LIN {X 0,Y 356.725,Z 687.983,A -85,B 0,C 180,E1 -20964.366,E2 -20964.366} C_VEL
LIN {X 0,Y 356.606,Z 693.356,A -85,B 0,C 180,E1 -20966.058,E2 -20966.058} C_VEL
LIN {X 0,Y 356.565,Z 697.608,A -85,B 0,C 180,E1 -20967.748,E2 -20967.748} C_VEL
LIN {X 0,Y 356.535,Z 699.927,A -85,B 0,C 180,E1 -20968.874,E2 -20968.874} C_VEL
LIN {X 0,Y 356.536,Z 701.836,A -85,B 0,C 180,E1 -20970,E2 -20970} C_VEL
LIN {X 0,Y 356.433,Z 704.456,A -85,B 0,C 180,E1 -20972.252,E2 -20972.252} C_VEL
LIN {X 0,Y 356.57,Z 705.616,A -85,B 0,C 180,E1 -20974.507,E2 -20974.507} C_VEL
LIN {X 0,Y 357.041,Z 705.356,A -85,B 0,C 180,E1 -20976.76,E2 -20976.76} C_VEL
LIN {X 0,Y 357.878,Z 703.692,A -85,B 0,C 180,E1 -20979.008,E2 -20979.008} C_VEL
LIN {X 0,Y 359.272,Z 700.612,A -85,B 0,C 180,E1 -20981.242,E2 -20981.242} C_VEL
LIN {X 0,Y 361.39,Z 696.021,A -85,B 0,C 180,E1 -20983.449,E2 -20983.449} C_VEL
LIN {X 0,Y 363.566,Z 690.094,A -85,B 0,C 180,E1 -20985.572,E2 -20985.572} C_VEL
LIN {X 0,Y 366.275,Z 682.97,A -85,B 0,C 180,E1 -20987.529,E2 -20987.529} C_VEL
LIN {X 0,Y 369.393,Z 674.484,A -85,B 0,C 180,E1 -20989.38,E2 -20989.38} C_VEL
LIN {X 0,Y 372.33,Z 665.799,A -85,B 0,C 180,E1 -20990.943,E2 -20990.943} C_VEL
LIN {X 0,Y 375.647,Z 655.443,A -85,B 0,C 180,E1 -20992.473,E2 -20992.473} C_VEL
LIN {X 0,Y 378.991,Z 644.123,A -85,B 0,C 180,E1 -20993.847,E2 -20993.847} C_VEL
LIN {X 0,Y 382.256,Z 631.813,A -85,B 0,C 180,E1 -20995.071,E2 -20995.071} C_VEL
LIN {X 0,Y 385.528,Z 618.219,A -85,B 0,C 180,E1 -20996.141,E2 -20996.141} C_VEL
LIN {X 0,Y 388.246,Z 605.333,A -85,B 0,C 180,E1 -20996.955,E2 -20996.955} C_VEL
LIN {X 0,Y 390.754,Z 591.419,A -85,B 0,C 180,E1 -20997.634,E2 -20997.634} C_VEL
LIN {X 0,Y 393.434,Z 571.086,A -85,B 0,C 180,E1 -20998.368,E2 -20998.368} C_VEL
LIN {X 0,Y 403.498,Z 492.971,A -85,B 0,C 180,E1 -21000.927,E2 -21000.927} C_VEL
LIN {X 0,Y 404.111,Z 486.973,A -85,B 0,C 180,E1 -21001.172,E2 -21001.172} C_VEL
LIN {X 0,Y 404.64,Z 471.101,A -85,B 0,C 180,E1 -21002.091,E2 -21002.091} C_VEL
LIN {X 0,Y 404.733,Z 459.98,A -85,B 0,C 180,E1 -21002.845,E2 -21002.845} C_VEL
LIN {X 0,Y 404.527,Z 444.365,A -85,B 0,C 180,E1 -21004.083,E2 -21004.083} C_VEL
LIN {X 0,Y 404.479,Z 437.616,A -85,B 0,C 180,E1 -21004.712,E2 -21004.712} C_VEL
LIN {X 0,Y 406.141,Z 430.503,A -85,B 0,C 180,E1 -21005.594,E2 -21005.594} C_VEL
LIN {X 0,Y 406.191,Z 429.05,A -85,B 0,C 180,E1 -21005.895,E2 -21005.895} C_VEL
LIN {X 0,Y 404.475,Z 426.255,A -85,B 0,C 180,E1 -21007.309,E2 -21007.309} C_VEL
LIN {X 0,Y 403.004,Z 424.19,A -85,B 0,C 180,E1 -21008.734,E2 -21008.734} C_VEL
LIN {X 0,Y 401.778,Z 422.799,A -85,B 0,C 180,E1 -21010.169,E2 -21010.169} C_VEL
LIN {X 0,Y 400.85,Z 422.022,A -85,B 0,C 180,E1 -21011.606,E2 -21011.606} C_VEL
LIN {X 0,Y 399.918,Z 421.946,A -85,B 0,C 180,E1 -21014.102,E2 -21014.102} C_VEL
LIN {X 0,Y 399.591,Z 423.06,A -85,B 0,C 180,E1 -21015.946,E2 -21015.946} C_VEL
LIN {X 0,Y 399.519,Z 425.806,A -85,B 0,C 180,E1 -21018.224,E2 -21018.224} C_VEL
LIN {X 0,Y 399.657,Z 428.065,A -85,B 0,C 180,E1 -21019.574,E2 -21019.574} C_VEL
LIN {X 0,Y 399.882,Z 432.504,A -85,B 0,C 180,E1 -21021.546,E2 -21021.546} C_VEL
LIN {X 0,Y 399.989,Z 438.039,A -85,B 0,C 180,E1 -21023.459,E2 -21023.459} C_VEL
LIN {X 0,Y 400.19,Z 440.153,A -85,B 0,C 180,E1 -21024.049,E2 -21024.049} C_VEL
LIN {X 0,Y 400.823,Z 442.858,A -85,B 0,C 180,E1 -21024.526,E2 -21024.526} C_VEL
LIN {X 0,Y 401.862,Z 457.626,A -85,B 0,C 180,E1 -21026.099,E2 -21026.099} C_VEL
LIN {X 0,Y 402.903,Z 473.385,A -85,B 0,C 180,E1 -21027.548,E2 -21027.548} C_VEL
LIN {X 0,Y 403.63,Z 486.988,A -85,B 0,C 180,E1 -21028.627,E2 -21028.627} C_VEL
LIN {X 0,Y 403.698,Z 493.511,A -85,B 0,C 180,E1 -21029.053,E2 -21029.053} C_VEL
LIN {X 0,Y 391.952,Z 585.206,A -85,B 0,C 180,E1 -21032.06,E2 -21032.06} C_VEL
LIN {X 0,Y 389.322,Z 600.595,A -85,B 0,C 180,E1 -21032.764,E2 -21032.764} C_VEL
LIN {X 0,Y 386.45,Z 614.844,A -85,B 0,C 180,E1 -21033.637,E2 -21033.637} C_VEL
LIN {X 0,Y 383.155,Z 628.608,A -85,B 0,C 180,E1 -21034.703,E2 -21034.703} C_VEL
LIN {X 0,Y 379.567,Z 642.265,A -85,B 0,C 180,E1 -21036.047,E2 -21036.047} C_VEL
LIN {X 0,Y 375.891,Z 654.552,A -85,B 0,C 180,E1 -21037.542,E2 -21037.542} C_VEL
LIN {X 0,Y 372.598,Z 664.764,A -85,B 0,C 180,E1 -21039.073,E2 -21039.073} C_VEL
LIN {X 0,Y 369.59,Z 673.378,A -85,B 0,C 180,E1 -21040.631,E2 -21040.631} C_VEL
LIN {X 0,Y 366.564,Z 681.749,A -85,B 0,C 180,E1 -21042.485,E2 -21042.485} C_VEL
LIN {X 0,Y 363.94,Z 688.565,A -85,B 0,C 180,E1 -21044.369,E2 -21044.369} C_VEL
LIN {X 0,Y 361.633,Z 694.693,A -85,B 0,C 180,E1 -21046.56,E2 -21046.56} C_VEL
LIN {X 0,Y 359.451,Z 699.244,A -85,B 0,C 180,E1 -21048.763,E2 -21048.763} C_VEL
LIN {X 0,Y 358.038,Z 702.291,A -85,B 0,C 180,E1 -21050.996,E2 -21050.996} C_VEL
LIN {X 0,Y 357.088,Z 703.936,A -85,B 0,C 180,E1 -21053.241,E2 -21053.241} C_VEL
LIN {X 0,Y 356.569,Z 704.185,A -85,B 0,C 180,E1 -21055.494,E2 -21055.494} C_VEL
LIN {X 0,Y 356.377,Z 703.027,A -85,B 0,C 180,E1 -21057.747,E2 -21057.747} C_VEL
LIN {X 0,Y 356.436,Z 700.429,A -85,B 0,C 180,E1 -21060,E2 -21060} C_VEL
LIN {X 0,Y 356.48,Z 696.249,A -85,B 0,C 180,E1 -21062.252,E2 -21062.252} C_VEL
LIN {X 0,Y 356.556,Z 692.048,A -85,B 0,C 180,E1 -21063.943,E2 -21063.943} C_VEL
LIN {X 0,Y 356.686,Z 685.768,A -85,B 0,C 180,E1 -21065.918,E2 -21065.918} C_VEL
LIN {X 0,Y 356.95,Z 677.854,A -85,B 0,C 180,E1 -21067.896,E2 -21067.896} C_VEL
LIN {X 0,Y 357.418,Z 669.599,A -85,B 0,C 180,E1 -21069.589,E2 -21069.589} C_VEL
LIN {X 0,Y 357.937,Z 659.637,A -85,B 0,C 180,E1 -21071.285,E2 -21071.285} C_VEL
LIN {X 0,Y 358.682,Z 648.682,A -85,B 0,C 180,E1 -21072.835,E2 -21072.835} C_VEL
LIN {X 0,Y 359.384,Z 636.555,A -85,B 0,C 180,E1 -21074.245,E2 -21074.245} C_VEL
LIN {X 0,Y 360.308,Z 623.272,A -85,B 0,C 180,E1 -21075.504,E2 -21075.504} C_VEL
LIN {X 0,Y 361.095,Z 609.51,A -85,B 0,C 180,E1 -21076.554,E2 -21076.554} C_VEL
LIN {X 0,Y 361.848,Z 594.748,A -85,B 0,C 180,E1 -21077.424,E2 -21077.424} C_VEL
LIN {X 0,Y 362.486,Z 579.344,A -85,B 0,C 180,E1 -21078.083,E2 -21078.083} C_VEL
LIN {X 0,Y 365.761,Z 475.035,A -85,B 0,C 180,E1 -21081.209,E2 -21081.209} C_VEL
LIN {X 0,Y 363.266,Z 445.339,A -85,B 0,C 180,E1 -21082.179,E2 -21082.179} C_VEL
LIN {X 0,Y 363.025,Z 439.566,A -85,B 0,C 180,E1 -21082.376,E2 -21082.376} C_VEL
LIN {X 0,Y 365.15,Z 412.697,A -85,B 0,C 180,E1 -21086.181,E2 -21086.181} C_VEL
LIN {X 0,Y 367.059,Z 389.753,A -85,B 0,C 180,E1 -21089.432,E2 -21089.432} C_VEL
LIN {X 0,Y 363.105,Z 371.527,A -85,B 0,C 180,E1 -21092.275,E2 -21092.275} C_VEL
LIN {X 0,Y 359.011,Z 353.326,A -85,B 0,C 180,E1 -21095.234,E2 -21095.234} C_VEL
LIN {X 0,Y 358.937,Z 353.332,A -85,B 0,C 180,E1 -21098.687,E2 -21098.687} C_VEL
LIN {X 0,Y 358.948,Z 353.327,A -85,B 0,C 180,E1 -21102.139,E2 -21102.139} C_VEL
LIN {X 0,Y 358.972,Z 353.324,A -85,B 0,C 180,E1 -21105.376,E2 -21105.376} C_VEL
LIN {X 0,Y 358.95,Z 353.33,A -85,B 0,C 180,E1 -21108.435,E2 -21108.435} C_VEL
LIN {X 0,Y 358.943,Z 353.33,A -85,B 0,C 180,E1 -21111.358,E2 -21111.358} C_VEL
LIN {X 0,Y 358.964,Z 353.328,A -85,B 0,C 180,E1 -21115.04,E2 -21115.04} C_VEL
LIN {X 0,Y 358.978,Z 353.321,A -85,B 0,C 180,E1 -21119.154,E2 -21119.154} C_VEL
LIN {X 0,Y 358.971,Z 353.327,A -85,B 0,C 180,E1 -21122.076,E2 -21122.076} C_VEL
LIN {X 0,Y 358.971,Z 353.329,A -85,B 0,C 180,E1 -21124.578,E2 -21124.578} C_VEL
LIN {X 0,Y 358.986,Z 353.325,A -85,B 0,C 180,E1 -21127.031,E2 -21127.031} C_VEL
LIN {X 0,Y 359.04,Z 353.321,A -85,B 0,C 180,E1 -21129.68,E2 -21129.68} C_VEL
LIN {X 0,Y 360.677,Z 357.57,A -85,B 0,C 180,E1 -21129.891,E2 -21129.891} C_VEL
LIN {X 0,Y 369.779,Z 378.619,A -85,B 0,C 180,E1 -21130.947,E2 -21130.947} C_VEL
LIN {X 0,Y 372.167,Z 384.575,A -85,B 0,C 180,E1 -21131.223,E2 -21131.223} C_VEL
LIN {X 0,Y 371.034,Z 437.953,A -85,B 0,C 180,E1 -21132.243,E2 -21132.243} C_VEL
LIN {X 0,Y 370.729,Z 471.673,A -85,B 0,C 180,E1 -21132.936,E2 -21132.936} C_VEL
LIN {X 0,Y 370.297,Z 486.255,A -85,B 0,C 180,E1 -21133.446,E2 -21133.446} C_VEL
LIN {X 0,Y 369.662,Z 499.54,A -85,B 0,C 180,E1 -21134.124,E2 -21134.124} C_VEL
LIN {X 0,Y 368.668,Z 512.538,A -85,B 0,C 180,E1 -21134.997,E2 -21134.997} C_VEL
LIN {X 0,Y 367.573,Z 525.068,A -85,B 0,C 180,E1 -21136.079,E2 -21136.079} C_VEL
LIN {X 0,Y 366.34,Z 537.468,A -85,B 0,C 180,E1 -21137.42,E2 -21137.42} C_VEL
LIN {X 0,Y 365.038,Z 546.962,A -85,B 0,C 180,E1 -21138.657,E2 -21138.657} C_VEL
LIN {X 0,Y 363.495,Z 557.369,A -85,B 0,C 180,E1 -21140.293,E2 -21140.293} C_VEL
LIN {X 0,Y 362.248,Z 565.948,A -85,B 0,C 180,E1 -21141.942,E2 -21141.942} C_VEL
LIN {X 0,Y 361.022,Z 574.183,A -85,B 0,C 180,E1 -21143.874,E2 -21143.874} C_VEL
LIN {X 0,Y 360.094,Z 579.941,A -85,B 0,C 180,E1 -21145.538,E2 -21145.538} C_VEL
LIN {X 0,Y 359.226,Z 586.093,A -85,B 0,C 180,E1 -21147.765,E2 -21147.765} C_VEL
LIN {X 0,Y 358.678,Z 590.642,A -85,B 0,C 180,E1 -21150,E2 -21150} C_VEL
LIN {X 0,Y 358.344,Z 593.75,A -85,B 0,C 180,E1 -21152.241,E2 -21152.241} C_VEL
LIN {X 0,Y 358.327,Z 595.525,A -85,B 0,C 180,E1 -21154.485,E2 -21154.485} C_VEL
LIN {X 0,Y 358.461,Z 596.018,A -85,B 0,C 180,E1 -21156.733,E2 -21156.733} C_VEL
LIN {X 0,Y 358.889,Z 595.216,A -85,B 0,C 180,E1 -21158.983,E2 -21158.983} C_VEL
LIN {X 0,Y 359.497,Z 593.109,A -85,B 0,C 180,E1 -21161.236,E2 -21161.236} C_VEL
LIN {X 0,Y 360.637,Z 589.599,A -85,B 0,C 180,E1 -21163.478,E2 -21163.478} C_VEL
LIN {X 0,Y 361.996,Z 584.607,A -85,B 0,C 180,E1 -21165.718,E2 -21165.718} C_VEL
LIN {X 0,Y 363.238,Z 579.74,A -85,B 0,C 180,E1 -21167.391,E2 -21167.391} C_VEL
LIN {X 0,Y 364.927,Z 572.832,A -85,B 0,C 180,E1 -21169.311,E2 -21169.311} C_VEL
LIN {X 0,Y 366.614,Z 565.377,A -85,B 0,C 180,E1 -21170.992,E2 -21170.992} C_VEL
LIN {X 0,Y 368.514,Z 556.498,A -85,B 0,C 180,E1 -21172.638,E2 -21172.638} C_VEL
LIN {X 0,Y 370.572,Z 545.708,A -85,B 0,C 180,E1 -21174.275,E2 -21174.275} C_VEL
LIN {X 0,Y 372.362,Z 534.709,A -85,B 0,C 180,E1 -21175.636,E2 -21175.636} C_VEL
LIN {X 0,Y 374.154,Z 522.52,A -85,B 0,C 180,E1 -21176.849,E2 -21176.849} C_VEL
LIN {X 0,Y 375.546,Z 510.75,A -85,B 0,C 180,E1 -21177.794,E2 -21177.794} C_VEL
LIN {X 0,Y 376.487,Z 499.1,A -85,B 0,C 180,E1 -21178.549,E2 -21178.549} C_VEL
LIN {X 0,Y 377.342,Z 484.813,A -85,B 0,C 180,E1 -21179.241,E2 -21179.241} C_VEL
LIN {X 0,Y 377.785,Z 470.873,A -85,B 0,C 180,E1 -21179.698,E2 -21179.698} C_VEL
LIN {X 0,Y 379.518,Z 405.514,A -85,B 0,C 180,E1 -21180.954,E2 -21180.954} C_VEL
LIN {X 0,Y 379.586,Z 394.59,A -85,B 0,C 180,E1 -21181.18,E2 -21181.18} C_VEL
LIN {X 0,Y 370.189,Z 374.863,A -85,B 0,C 180,E1 -21182.424,E2 -21182.424} C_VEL
LIN {X 0,Y 360.343,Z 356.812,A -85,B 0,C 180,E1 -21183.757,E2 -21183.757} C_VEL
LIN {X 0,Y 359.066,Z 354.304,A -85,B 0,C 180,E1 -21183.941,E2 -21183.941} C_VEL
LIN {X 0,Y 358.893,Z 353.337,A -85,B 0,C 180,E1 -21184.001,E2 -21184.001} C_VEL
LIN {X 0,Y 358.912,Z 353.335,A -85,B 0,C 180,E1 -21187.228,E2 -21187.228} C_VEL
LIN {X 0,Y 358.912,Z 353.338,A -85,B 0,C 180,E1 -21190.437,E2 -21190.437} C_VEL
LIN {X 0,Y 358.886,Z 353.338,A -85,B 0,C 180,E1 -21191.966,E2 -21191.966} C_VEL
LIN {X 0,Y 358.237,Z 353.422,A -85,B 0,C 180,E1 -21192.901,E2 -21192.901} C_VEL
LIN {X 0,Y 355.372,Z 353.774,A -85,B 0,C 180,E1 -21194.422,E2 -21194.422} C_VEL
LIN {X 0,Y 352.944,Z 354.077,A -85,B 0,C 180,E1 -21195.653,E2 -21195.653} C_VEL
LIN {X 0,Y 351.92,Z 354.207,A -85,B 0,C 180,E1 -21196.606,E2 -21196.606} C_VEL
LIN {X 0,Y 351.848,Z 354.209,A -85,B 0,C 180,E1 -21196.929,E2 -21196.929} C_VEL
LIN {X 0,Y 351.854,Z 354.209,A -85,B 0,C 180,E1 -21200.429,E2 -21200.429} C_VEL
LIN {X 0,Y 351.864,Z 354.168,A -85,B 0,C 180,E1 -21203.33,E2 -21203.33} C_VEL
LIN {X 0,Y 351.865,Z 354.208,A -85,B 0,C 180,E1 -21206.729,E2 -21206.729} C_VEL
LIN {X 0,Y 351.886,Z 354.2,A -85,B 0,C 180,E1 -21210.156,E2 -21210.156} C_VEL
LIN {X 0,Y 351.946,Z 354.189,A -85,B 0,C 180,E1 -21214.033,E2 -21214.033} C_VEL
LIN {X 0,Y 351.954,Z 354.198,A -85,B 0,C 180,E1 -21217.572,E2 -21217.572} C_VEL
LIN {X 0,Y 358.141,Z 377.526,A -85,B 0,C 180,E1 -21218.454,E2 -21218.454} C_VEL
LIN {X 0,Y 355.675,Z 470.004,A -85,B 0,C 180,E1 -21221.237,E2 -21221.237} C_VEL
LIN {X 0,Y 355.334,Z 485.438,A -85,B 0,C 180,E1 -21221.912,E2 -21221.912} C_VEL
LIN {X 0,Y 354.727,Z 501.095,A -85,B 0,C 180,E1 -21222.845,E2 -21222.845} C_VEL
LIN {X 0,Y 354.11,Z 514.993,A -85,B 0,C 180,E1 -21223.923,E2 -21223.923} C_VEL
LIN {X 0,Y 353.351,Z 528.412,A -85,B 0,C 180,E1 -21225.213,E2 -21225.213} C_VEL
LIN {X 0,Y 352.707,Z 540.9,A -85,B 0,C 180,E1 -21226.681,E2 -21226.681} C_VEL
LIN {X 0,Y 352.08,Z 551.828,A -85,B 0,C 180,E1 -21228.233,E2 -21228.233} C_VEL
LIN {X 0,Y 351.512,Z 561.982,A -85,B 0,C 180,E1 -21229.958,E2 -21229.958} C_VEL
LIN {X 0,Y 351.108,Z 570.476,A -85,B 0,C 180,E1 -21231.684,E2 -21231.684} C_VEL
LIN {X 0,Y 350.843,Z 578.663,A -85,B 0,C 180,E1 -21233.696,E2 -21233.696} C_VEL
LIN {X 0,Y 350.805,Z 584.378,A -85,B 0,C 180,E1 -21235.419,E2 -21235.419} C_VEL
LIN {X 0,Y 350.847,Z 589.454,A -85,B 0,C 180,E1 -21237.294,E2 -21237.294} C_VEL
LIN {X 0,Y 351.077,Z 593.911,A -85,B 0,C 180,E1 -21239.428,E2 -21239.428} C_VEL
LIN {X 0,Y 351.487,Z 596.487,A -85,B 0,C 180,E1 -21241.142,E2 -21241.142} C_VEL
LIN {X 0,Y 352.352,Z 598.709,A -85,B 0,C 180,E1 -21243.419,E2 -21243.419} C_VEL
LIN {X 0,Y 353.573,Z 599.494,A -85,B 0,C 180,E1 -21245.684,E2 -21245.684} C_VEL
LIN {X 0,Y 355.059,Z 598.85,A -85,B 0,C 180,E1 -21247.937,E2 -21247.937} C_VEL
LIN {X 0,Y 357.111,Z 596.776,A -85,B 0,C 180,E1 -21250.167,E2 -21250.167} C_VEL
LIN {X 0,Y 359.825,Z 593.175,A -85,B 0,C 180,E1 -21252.364,E2 -21252.364} C_VEL
LIN {X 0,Y 361.983,Z 589.458,A -85,B 0,C 180,E1 -21253.997,E2 -21253.997} C_VEL
LIN {X 0,Y 365.123,Z 583.078,A -85,B 0,C 180,E1 -21256.15,E2 -21256.15} C_VEL
LIN {X 0,Y 368.201,Z 575.99,A -85,B 0,C 180,E1 -21257.978,E2 -21257.978} C_VEL
LIN {X 0,Y 371.607,Z 566.998,A -85,B 0,C 180,E1 -21259.833,E2 -21259.833} C_VEL
LIN {X 0,Y 374.756,Z 557.748,A -85,B 0,C 180,E1 -21261.375,E2 -21261.375} C_VEL
LIN {X 0,Y 378.134,Z 546.581,A -85,B 0,C 180,E1 -21262.892,E2 -21262.892} C_VEL
LIN {X 0,Y 381.462,Z 534.045,A -85,B 0,C 180,E1 -21264.258,E2 -21264.258} C_VEL
LIN {X 0,Y 384.193,Z 521.641,A -85,B 0,C 180,E1 -21265.368,E2 -21265.368} C_VEL
LIN {X 0,Y 386.585,Z 508.111,A -85,B 0,C 180,E1 -21266.353,E2 -21266.353} C_VEL
LIN {X 0,Y 388.641,Z 493.528,A -85,B 0,C 180,E1 -21267.179,E2 -21267.179} C_VEL
LIN {X 0,Y 390.48,Z 476.072,A -85,B 0,C 180,E1 -21267.909,E2 -21267.909} C_VEL
LIN {X 0,Y 394.84,Z 439.615,A -85,B 0,C 180,E1 -21269.138,E2 -21269.138} C_VEL
LIN {X 0,Y 397.763,Z 417.256,A -85,B 0,C 180,E1 -21269.877,E2 -21269.877} C_VEL
LIN {X 0,Y 394.545,Z 410.848,A -85,B 0,C 180,E1 -21271.112,E2 -21271.112} C_VEL
LIN {X 0,Y 391.131,Z 404.658,A -85,B 0,C 180,E1 -21272.567,E2 -21272.567} C_VEL
LIN {X 0,Y 389.244,Z 401.397,A -85,B 0,C 180,E1 -21273.486,E2 -21273.486} C_VEL
LIN {X 0,Y 386.985,Z 397.73,A -85,B 0,C 180,E1 -21274.686,E2 -21274.686} C_VEL
LIN {X 0,Y 384.579,Z 393.864,A -85,B 0,C 180,E1 -21276.183,E2 -21276.183} C_VEL
LIN {X 0,Y 382.361,Z 390.848,A -85,B 0,C 180,E1 -21277.858,E2 -21277.858} C_VEL
LIN {X 0,Y 381.655,Z 389.329,A -85,B 0,C 180,E1 -21278.608,E2 -21278.608} C_VEL
LIN {X 0,Y 379.403,Z 387.476,A -85,B 0,C 180,E1 -21281.653,E2 -21281.653} C_VEL
LIN {X 0,Y 379.063,Z 387.134,A -85,B 0,C 180,E1 -21283.891,E2 -21283.891} C_VEL
LIN {X 0,Y 379.695,Z 387.952,A -85,B 0,C 180,E1 -21286.009,E2 -21286.009} C_VEL
LIN {X 0,Y 381.505,Z 389.601,A -85,B 0,C 180,E1 -21288.266,E2 -21288.266} C_VEL
LIN {X 0,Y 383.095,Z 392.706,A -85,B 0,C 180,E1 -21289.849,E2 -21289.849} C_VEL
LIN {X 0,Y 384.649,Z 394.585,A -85,B 0,C 180,E1 -21290.94,E2 -21290.94} C_VEL
LIN {X 0,Y 385.11,Z 396.18,A -85,B 0,C 180,E1 -21291.344,E2 -21291.344} C_VEL
LIN {X 0,Y 386.64,Z 403.777,A -85,B 0,C 180,E1 -21292.794,E2 -21292.794} C_VEL
LIN {X 0,Y 389.443,Z 417.992,A -85,B 0,C 180,E1 -21294.984,E2 -21294.984} C_VEL
LIN {X 0,Y 389.605,Z 422.458,A -85,B 0,C 180,E1 -21295.388,E2 -21295.388} C_VEL
LIN {X 0,Y 390.1,Z 441.215,A -85,B 0,C 180,E1 -21296.884,E2 -21296.884} C_VEL
LIN {X 0,Y 390.469,Z 462.05,A -85,B 0,C 180,E1 -21298.323,E2 -21298.323} C_VEL
LIN {X 0,Y 390.358,Z 475.663,A -85,B 0,C 180,E1 -21299.13,E2 -21299.13} C_VEL
LIN {X 0,Y 389.701,Z 489.992,A -85,B 0,C 180,E1 -21299.817,E2 -21299.817} C_VEL
LIN {X 0,Y 383.661,Z 539.895,A -85,B 0,C 180,E1 -21301.475,E2 -21301.475} C_VEL
LIN {X 0,Y 380.891,Z 555.484,A -85,B 0,C 180,E1 -21302.146,E2 -21302.146} C_VEL
LIN {X 0,Y 377.711,Z 570.021,A -85,B 0,C 180,E1 -21302.977,E2 -21302.977} C_VEL
LIN {X 0,Y 373.554,Z 586.152,A -85,B 0,C 180,E1 -21304.153,E2 -21304.153} C_VEL
LIN {X 0,Y 369.789,Z 599.191,A -85,B 0,C 180,E1 -21305.372,E2 -21305.372} C_VEL
LIN {X 0,Y 366.374,Z 610.138,A -85,B 0,C 180,E1 -21306.627,E2 -21306.627} C_VEL
LIN {X 0,Y 362.633,Z 621.676,A -85,B 0,C 180,E1 -21308.234,E2 -21308.234} C_VEL
LIN {X 0,Y 359.212,Z 632.199,A -85,B 0,C 180,E1 -21310.047,E2 -21310.047} C_VEL
LIN {X 0,Y 356.141,Z 641.2,A -85,B 0,C 180,E1 -21311.955,E2 -21311.955} C_VEL
LIN {X 0,Y 353.827,Z 648.647,A -85,B 0,C 180,E1 -21313.91,E2 -21313.91} C_VEL
LIN {X 0,Y 351.965,Z 655.474,A -85,B 0,C 180,E1 -21316.183,E2 -21316.183} C_VEL
LIN {X 0,Y 350.749,Z 660.764,A -85,B 0,C 180,E1 -21318.48,E2 -21318.48} C_VEL
LIN {X 0,Y 350.609,Z 661.973,A -85,B 0,C 180,E1 -21319.059,E2 -21319.059} C_VEL
LIN {X 0,Y 350.177,Z 671.911,A -85,B 0,C 180,E1 -21320.792,E2 -21320.792} C_VEL
LIN {X 0,Y 349.799,Z 680.094,A -85,B 0,C 180,E1 -21322.521,E2 -21322.521} C_VEL
LIN {X 0,Y 349.661,Z 686.861,A -85,B 0,C 180,E1 -21324.251,E2 -21324.251} C_VEL
LIN {X 0,Y 349.56,Z 692.399,A -85,B 0,C 180,E1 -21325.978,E2 -21325.978} C_VEL
LIN {X 0,Y 349.498,Z 696.863,A -85,B 0,C 180,E1 -21327.703,E2 -21327.703} C_VEL
LIN {X 0,Y 349.454,Z 700.358,A -85,B 0,C 180,E1 -21329.426,E2 -21329.426} C_VEL
LIN {X 0,Y 349.373,Z 702.903,A -85,B 0,C 180,E1 -21331.149,E2 -21331.149} C_VEL
LIN {X 0,Y 349.378,Z 705.024,A -85,B 0,C 180,E1 -21333.448,E2 -21333.448} C_VEL
LIN {X 0,Y 349.708,Z 705.692,A -85,B 0,C 180,E1 -21335.747,E2 -21335.747} C_VEL
LIN {X 0,Y 350.41,Z 704.936,A -85,B 0,C 180,E1 -21338.043,E2 -21338.043} C_VEL
LIN {X 0,Y 351.518,Z 702.787,A -85,B 0,C 180,E1 -21340.331,E2 -21340.331} C_VEL
LIN {X 0,Y 353.358,Z 699.197,A -85,B 0,C 180,E1 -21342.594,E2 -21342.594} C_VEL
LIN {X 0,Y 355.677,Z 694.096,A -85,B 0,C 180,E1 -21344.833,E2 -21344.833} C_VEL
LIN {X 0,Y 357.621,Z 689.234,A -85,B 0,C 180,E1 -21346.499,E2 -21346.499} C_VEL
LIN {X 0,Y 360.976,Z 681.121,A -85,B 0,C 180,E1 -21348.673,E2 -21348.673} C_VEL
LIN {X 0,Y 364.363,Z 672.316,A -85,B 0,C 180,E1 -21350.538,E2 -21350.538} C_VEL
LIN {X 0,Y 367.641,Z 663.241,A -85,B 0,C 180,E1 -21352.104,E2 -21352.104} C_VEL
LIN {X 0,Y 371.549,Z 651.413,A -85,B 0,C 180,E1 -21353.763,E2 -21353.763} C_VEL
LIN {X 0,Y 375.196,Z 639.346,A -85,B 0,C 180,E1 -21355.133,E2 -21355.133} C_VEL
LIN {X 0,Y 378.422,Z 627.589,A -85,B 0,C 180,E1 -21356.226,E2 -21356.226} C_VEL
LIN {X 0,Y 381.863,Z 613.173,A -85,B 0,C 180,E1 -21357.295,E2 -21357.295} C_VEL
LIN {X 0,Y 385.061,Z 597.984,A -85,B 0,C 180,E1 -21358.152,E2 -21358.152} C_VEL
LIN {X 0,Y 387.515,Z 583.341,A -85,B 0,C 180,E1 -21358.767,E2 -21358.767} C_VEL
LIN {X 0,Y 399.954,Z 491.497,A -85,B 0,C 180,E1 -21361.846,E2 -21361.846} C_VEL
LIN {X 0,Y 400.582,Z 481.749,A -85,B 0,C 180,E1 -21362.367,E2 -21362.367} C_VEL
LIN {X 0,Y 401.101,Z 466.574,A -85,B 0,C 180,E1 -21363.339,E2 -21363.339} C_VEL
LIN {X 0,Y 401.201,Z 449.322,A -85,B 0,C 180,E1 -21364.695,E2 -21364.695} C_VEL
LIN {X 0,Y 401.22,Z 437.905,A -85,B 0,C 180,E1 -21365.776,E2 -21365.776} C_VEL
LIN {X 0,Y 401.735,Z 435.888,A -85,B 0,C 180,E1 -21366.039,E2 -21366.039} C_VEL
LIN {X 0,Y 401.941,Z 434.259,A -85,B 0,C 180,E1 -21366.335,E2 -21366.335} C_VEL
LIN {X 0,Y 400.008,Z 431.305,A -85,B 0,C 180,E1 -21368.003,E2 -21368.003} C_VEL
LIN {X 0,Y 398.697,Z 429.59,A -85,B 0,C 180,E1 -21369.375,E2 -21369.375} C_VEL
LIN {X 0,Y 397.615,Z 428.454,A -85,B 0,C 180,E1 -21370.756,E2 -21370.756} C_VEL
LIN {X 0,Y 396.75,Z 427.877,A -85,B 0,C 180,E1 -21372.142,E2 -21372.142} C_VEL
LIN {X 0,Y 396.126,Z 427.794,A -85,B 0,C 180,E1 -21373.599,E2 -21373.599} C_VEL
LIN {X 0,Y 395.735,Z 428.344,A -85,B 0,C 180,E1 -21375.072,E2 -21375.072} C_VEL
LIN {X 0,Y 395.476,Z 429.583,A -85,B 0,C 180,E1 -21376.566,E2 -21376.566} C_VEL
LIN {X 0,Y 395.364,Z 432.992,A -85,B 0,C 180,E1 -21379.042,E2 -21379.042} C_VEL
LIN {X 0,Y 395.429,Z 437.508,A -85,B 0,C 180,E1 -21381.205,E2 -21381.205} C_VEL
LIN {X 0,Y 395.627,Z 440.106,A -85,B 0,C 180,E1 -21382.136,E2 -21382.136} C_VEL
LIN {X 0,Y 397.718,Z 446.772,A -85,B 0,C 180,E1 -21383.775,E2 -21383.775} C_VEL
LIN {X 0,Y 398.279,Z 457.122,A -85,B 0,C 180,E1 -21384.94,E2 -21384.94} C_VEL
LIN {X 0,Y 399.104,Z 473.805,A -85,B 0,C 180,E1 -21386.57,E2 -21386.57} C_VEL
LIN {X 0,Y 399.675,Z 488.703,A -85,B 0,C 180,E1 -21387.798,E2 -21387.798} C_VEL
LIN {X 0,Y 399.696,Z 495.123,A -85,B 0,C 180,E1 -21388.24,E2 -21388.24} C_VEL
LIN {X 0,Y 387.55,Z 584.975,A -85,B 0,C 180,E1 -21391.236,E2 -21391.236} C_VEL
LIN {X 0,Y 384.897,Z 599.742,A -85,B 0,C 180,E1 -21391.909,E2 -21391.909} C_VEL
LIN {X 0,Y 382.031,Z 613.198,A -85,B 0,C 180,E1 -21392.718,E2 -21392.718} C_VEL
LIN {X 0,Y 378.607,Z 627.223,A -85,B 0,C 180,E1 -21393.788,E2 -21393.788} C_VEL
LIN {X 0,Y 375.071,Z 639.894,A -85,B 0,C 180,E1 -21395.006,E2 -21395.006} C_VEL
LIN {X 0,Y 371.498,Z 651.579,A -85,B 0,C 180,E1 -21396.381,E2 -21396.381} C_VEL
LIN {X 0,Y 367.889,Z 662.278,A -85,B 0,C 180,E1 -21397.912,E2 -21397.912} C_VEL
LIN {X 0,Y 364.636,Z 671.25,A -85,B 0,C 180,E1 -21399.478,E2 -21399.478} C_VEL
LIN {X 0,Y 361.278,Z 679.963,A -85,B 0,C 180,E1 -21401.343,E2 -21401.343} C_VEL
LIN {X 0,Y 358.718,Z 686.184,A -85,B 0,C 180,E1 -21402.969,E2 -21402.969} C_VEL
LIN {X 0,Y 356.487,Z 691.34,A -85,B 0,C 180,E1 -21404.618,E2 -21404.618} C_VEL
LIN {X 0,Y 354.167,Z 696.786,A -85,B 0,C 180,E1 -21406.854,E2 -21406.854} C_VEL
LIN {X 0,Y 352.531,Z 699.841,A -85,B 0,C 180,E1 -21408.54,E2 -21408.54} C_VEL
LIN {X 0,Y 351.022,Z 702.673,A -85,B 0,C 180,E1 -21410.815,E2 -21410.815} C_VEL
LIN {X 0,Y 350.039,Z 704.106,A -85,B 0,C 180,E1 -21413.105,E2 -21413.105} C_VEL
LIN {X 0,Y 349.483,Z 704.148,A -85,B 0,C 180,E1 -21415.402,E2 -21415.402} C_VEL
LIN {X 0,Y 349.291,Z 702.764,A -85,B 0,C 180,E1 -21417.702,E2 -21417.702} C_VEL
LIN {X 0,Y 349.356,Z 699.926,A -85,B 0,C 180,E1 -21420,E2 -21420} C_VEL
LIN {X 0,Y 349.395,Z 696.826,A -85,B 0,C 180,E1 -21421.724,E2 -21421.724} C_VEL
LIN {X 0,Y 349.442,Z 692.719,A -85,B 0,C 180,E1 -21423.448,E2 -21423.448} C_VEL
LIN {X 0,Y 349.57,Z 687.607,A -85,B 0,C 180,E1 -21425.174,E2 -21425.174} C_VEL
LIN {X 0,Y 349.81,Z 680.21,A -85,B 0,C 180,E1 -21427.19,E2 -21427.19} C_VEL
LIN {X 0,Y 350.123,Z 672.424,A -85,B 0,C 180,E1 -21428.92,E2 -21428.92} C_VEL
LIN {X 0,Y 350.669,Z 663.069,A -85,B 0,C 180,E1 -21430.648,E2 -21430.648} C_VEL
LIN {X 0,Y 351.368,Z 652.325,A -85,B 0,C 180,E1 -21432.29,E2 -21432.29} C_VEL
LIN {X 0,Y 352.098,Z 640.244,A -85,B 0,C 180,E1 -21433.811,E2 -21433.811} C_VEL
LIN {X 0,Y 352.88,Z 627.823,A -85,B 0,C 180,E1 -21435.101,E2 -21435.101} C_VEL
LIN {X 0,Y 353.786,Z 614.357,A -85,B 0,C 180,E1 -21436.24,E2 -21436.24} C_VEL
LIN {X 0,Y 354.433,Z 600.335,A -85,B 0,C 180,E1 -21437.17,E2 -21437.17} C_VEL
LIN {X 0,Y 355.117,Z 585.482,A -85,B 0,C 180,E1 -21437.914,E2 -21437.914} C_VEL
LIN {X 0,Y 355.72,Z 568.346,A -85,B 0,C 180,E1 -21438.508,E2 -21438.508} C_VEL
LIN {X 0,Y 358.743,Z 475.397,A -85,B 0,C 180,E1 -21441.363,E2 -21441.363} C_VEL
LIN {X 0,Y 356.26,Z 445.66,A -85,B 0,C 180,E1 -21442.355,E2 -21442.355} C_VEL
LIN {X 0,Y 356.016,Z 439.606,A -85,B 0,C 180,E1 -21442.563,E2 -21442.563} C_VEL
LIN {X 0,Y 358.22,Z 412.54,A -85,B 0,C 180,E1 -21446.448,E2 -21446.448} C_VEL
LIN {X 0,Y 360.065,Z 390.739,A -85,B 0,C 180,E1 -21449.58,E2 -21449.58} C_VEL
LIN {X 0,Y 355.778,Z 371.172,A -85,B 0,C 180,E1 -21452.684,E2 -21452.684} C_VEL
LIN {X 0,Y 351.972,Z 354.202,A -85,B 0,C 180,E1 -21455.453,E2 -21455.453} C_VEL
LIN {X 0,Y 351.874,Z 354.214,A -85,B 0,C 180,E1 -21459.074,E2 -21459.074} C_VEL
LIN {X 0,Y 351.923,Z 354.203,A -85,B 0,C 180,E1 -21462.588,E2 -21462.588} C_VEL
LIN {X 0,Y 351.939,Z 354.198,A -85,B 0,C 180,E1 -21465.846,E2 -21465.846} C_VEL
LIN {X 0,Y 351.882,Z 354.206,A -85,B 0,C 180,E1 -21469.15,E2 -21469.15} C_VEL
LIN {X 0,Y 351.914,Z 354.205,A -85,B 0,C 180,E1 -21472.765,E2 -21472.765} C_VEL
LIN {X 0,Y 351.895,Z 354.207,A -85,B 0,C 180,E1 -21476.128,E2 -21476.128} C_VEL
LIN {X 0,Y 351.928,Z 354.201,A -85,B 0,C 180,E1 -21480.16,E2 -21480.16} C_VEL
LIN {X 0,Y 351.931,Z 354.203,A -85,B 0,C 180,E1 -21483.591,E2 -21483.591} C_VEL
LIN {X 0,Y 351.98,Z 354.201,A -85,B 0,C 180,E1 -21486.547,E2 -21486.547} C_VEL
LIN {X 0,Y 351.979,Z 354.2,A -85,B 0,C 180,E1 -21489.191,E2 -21489.191} C_VEL
LIN {X 0,Y 352.975,Z 357.048,A -85,B 0,C 180,E1 -21489.329,E2 -21489.329} C_VEL
LIN {X 0,Y 361.343,Z 375.884,A -85,B 0,C 180,E1 -21490.327,E2 -21490.327} C_VEL
LIN {X 0,Y 365.602,Z 386.378,A -85,B 0,C 180,E1 -21490.834,E2 -21490.834} C_VEL
LIN {X 0,Y 364.181,Z 459.074,A -85,B 0,C 180,E1 -21492.258,E2 -21492.258} C_VEL
LIN {X 0,Y 363.992,Z 476.544,A -85,B 0,C 180,E1 -21492.682,E2 -21492.682} C_VEL
LIN {X 0,Y 363.496,Z 490.484,A -85,B 0,C 180,E1 -21493.235,E2 -21493.235} C_VEL
LIN {X 0,Y 362.641,Z 504.553,A -85,B 0,C 180,E1 -21494.024,E2 -21494.024} C_VEL
LIN {X 0,Y 361.565,Z 517.456,A -85,B 0,C 180,E1 -21494.983,E2 -21494.983} C_VEL
LIN {X 0,Y 360.382,Z 530.434,A -85,B 0,C 180,E1 -21496.226,E2 -21496.226} C_VEL
LIN {X 0,Y 359.032,Z 542.099,A -85,B 0,C 180,E1 -21497.608,E2 -21497.608} C_VEL
LIN {X 0,Y 357.617,Z 551.792,A -85,B 0,C 180,E1 -21498.991,E2 -21498.991} C_VEL
LIN {X 0,Y 356.174,Z 561.456,A -85,B 0,C 180,E1 -21500.663,E2 -21500.663} C_VEL
LIN {X 0,Y 354.949,Z 569.479,A -85,B 0,C 180,E1 -21502.345,E2 -21502.345} C_VEL
LIN {X 0,Y 353.696,Z 577.173,A -85,B 0,C 180,E1 -21504.318,E2 -21504.318} C_VEL
LIN {X 0,Y 352.853,Z 582.567,A -85,B 0,C 180,E1 -21506.016,E2 -21506.016} C_VEL
LIN {X 0,Y 352.01,Z 588.238,A -85,B 0,C 180,E1 -21508.29,E2 -21508.29} C_VEL
LIN {X 0,Y 351.642,Z 591.497,A -85,B 0,C 180,E1 -21510,E2 -21510} C_VEL
LIN {X 0,Y 351.277,Z 594.576,A -85,B 0,C 180,E1 -21512.286,E2 -21512.286} C_VEL
LIN {X 0,Y 351.278,Z 596.317,A -85,B 0,C 180,E1 -21514.575,E2 -21514.575} C_VEL
LIN {X 0,Y 351.438,Z 596.778,A -85,B 0,C 180,E1 -21516.868,E2 -21516.868} C_VEL
LIN {X 0,Y 351.892,Z 595.945,A -85,B 0,C 180,E1 -21519.163,E2 -21519.163} C_VEL
LIN {X 0,Y 352.535,Z 593.807,A -85,B 0,C 180,E1 -21521.46,E2 -21521.46} C_VEL
LIN {X 0,Y 353.717,Z 590.264,A -85,B 0,C 180,E1 -21523.747,E2 -21523.747} C_VEL
LIN {X 0,Y 355.174,Z 585.233,A -85,B 0,C 180,E1 -21526.028,E2 -21526.028} C_VEL
LIN {X 0,Y 356.463,Z 580.328,A -85,B 0,C 180,E1 -21527.733,E2 -21527.733} C_VEL
LIN {X 0,Y 358.252,Z 573.283,A -85,B 0,C 180,E1 -21529.711,E2 -21529.711} C_VEL
LIN {X 0,Y 359.971,Z 565.875,A -85,B 0,C 180,E1 -21531.398,E2 -21531.398} C_VEL
LIN {X 0,Y 361.954,Z 556.941,A -85,B 0,C 180,E1 -21533.071,E2 -21533.071} C_VEL
LIN {X 0,Y 364.099,Z 546.084,A -85,B 0,C 180,E1 -21534.735,E2 -21534.735} C_VEL
LIN {X 0,Y 365.953,Z 534.984,A -85,B 0,C 180,E1 -21536.119,E2 -21536.119} C_VEL
LIN {X 0,Y 367.831,Z 522.648,A -85,B 0,C 180,E1 -21537.349,E2 -21537.349} C_VEL
LIN {X 0,Y 369.22,Z 510.712,A -85,B 0,C 180,E1 -21538.312,E2 -21538.312} C_VEL
LIN {X 0,Y 370.227,Z 498.868,A -85,B 0,C 180,E1 -21539.078,E2 -21539.078} C_VEL
LIN {X 0,Y 371.056,Z 485.349,A -85,B 0,C 180,E1 -21539.732,E2 -21539.732} C_VEL
LIN {X 0,Y 371.507,Z 471.799,A -85,B 0,C 180,E1 -21540.184,E2 -21540.184} C_VEL
LIN {X 0,Y 373.057,Z 414.014,A -85,B 0,C 180,E1 -21541.318,E2 -21541.318} C_VEL
LIN {X 0,Y 373.529,Z 397.579,A -85,B 0,C 180,E1 -21541.633,E2 -21541.633} C_VEL
LIN {X 0,Y 372.343,Z 394.341,A -85,B 0,C 180,E1 -21541.806,E2 -21541.806} C_VEL
LIN {X 0,Y 363.162,Z 375.511,A -85,B 0,C 180,E1 -21543.06,E2 -21543.06} C_VEL
LIN {X 0,Y 353.104,Z 357.398,A -85,B 0,C 180,E1 -21544.47,E2 -21544.47} C_VEL
LIN {X 0,Y 351.936,Z 354.742,A -85,B 0,C 180,E1 -21544.654,E2 -21544.654} C_VEL
LIN {X 0,Y 351.87,Z 354.212,A -85,B 0,C 180,E1 -21544.7,E2 -21544.7} C_VEL
LIN {X 0,Y 351.839,Z 354.216,A -85,B 0,C 180,E1 -21548.109,E2 -21548.109} C_VEL
LIN {X 0,Y 351.852,Z 354.218,A -85,B 0,C 180,E1 -21551.068,E2 -21551.068} C_VEL
LIN {X 0,Y 351.872,Z 354.211,A -85,B 0,C 180,E1 -21554.223,E2 -21554.223} C_VEL
LIN {X 0,Y 351.848,Z 354.209,A -85,B 0,C 180,E1 -21556.929,E2 -21556.929} C_VEL
LIN {X 0,Y 351.2,Z 354.294,A -85,B 0,C 180,E1 -21557.884,E2 -21557.884} C_VEL
LIN {X 0,Y 348.328,Z 354.653,A -85,B 0,C 180,E1 -21559.437,E2 -21559.437} C_VEL
LIN {X 0,Y 345.89,Z 354.95,A -85,B 0,C 180,E1 -21560.695,E2 -21560.695} C_VEL
LIN {X 0,Y 344.859,Z 355.058,A -85,B 0,C 180,E1 -21561.668,E2 -21561.668} C_VEL
LIN {X 0,Y 344.784,Z 355.059,A -85,B 0,C 180,E1 -21561.998,E2 -21561.998} C_VEL
LIN {X 0,Y 344.81,Z 355.071,A -85,B 0,C 180,E1 -21565.334,E2 -21565.334} C_VEL
LIN {X 0,Y 344.816,Z 355.081,A -85,B 0,C 180,E1 -21568.559,E2 -21568.559} C_VEL
LIN {X 0,Y 344.839,Z 355.085,A -85,B 0,C 180,E1 -21572.148,E2 -21572.148} C_VEL
LIN {X 0,Y 344.863,Z 355.074,A -85,B 0,C 180,E1 -21574.752,E2 -21574.752} C_VEL
LIN {X 0,Y 344.907,Z 355.078,A -85,B 0,C 180,E1 -21577.417,E2 -21577.417} C_VEL
LIN {X 0,Y 351.041,Z 378.111,A -85,B 0,C 180,E1 -21578.309,E2 -21578.309} C_VEL
LIN {X 0,Y 348.578,Z 471.546,A -85,B 0,C 180,E1 -21581.208,E2 -21581.208} C_VEL
LIN {X 0,Y 348.209,Z 486.888,A -85,B 0,C 180,E1 -21581.908,E2 -21581.908} C_VEL
LIN {X 0,Y 347.578,Z 502.301,A -85,B 0,C 180,E1 -21582.859,E2 -21582.859} C_VEL
LIN {X 0,Y 346.911,Z 516.892,A -85,B 0,C 180,E1 -21584.032,E2 -21584.032} C_VEL
LIN {X 0,Y 346.143,Z 530.121,A -85,B 0,C 180,E1 -21585.348,E2 -21585.348} C_VEL
LIN {X 0,Y 345.601,Z 541.383,A -85,B 0,C 180,E1 -21586.703,E2 -21586.703} C_VEL
LIN {X 0,Y 344.95,Z 552.358,A -85,B 0,C 180,E1 -21588.284,E2 -21588.284} C_VEL
LIN {X 0,Y 344.391,Z 562.549,A -85,B 0,C 180,E1 -21590.044,E2 -21590.044} C_VEL
LIN {X 0,Y 343.994,Z 571.085,A -85,B 0,C 180,E1 -21591.805,E2 -21591.805} C_VEL
LIN {X 0,Y 343.734,Z 579.332,A -85,B 0,C 180,E1 -21593.858,E2 -21593.858} C_VEL
LIN {X 0,Y 343.736,Z 585.971,A -85,B 0,C 180,E1 -21595.91,E2 -21595.91} C_VEL
LIN {X 0,Y 343.785,Z 590.543,A -85,B 0,C 180,E1 -21597.664,E2 -21597.664} C_VEL
LIN {X 0,Y 343.991,Z 594.181,A -85,B 0,C 180,E1 -21599.416,E2 -21599.416} C_VEL
LIN {X 0,Y 344.408,Z 596.979,A -85,B 0,C 180,E1 -21601.165,E2 -21601.165} C_VEL
LIN {X 0,Y 345.328,Z 599.41,A -85,B 0,C 180,E1 -21603.488,E2 -21603.488} C_VEL
LIN {X 0,Y 346.584,Z 600.444,A -85,B 0,C 180,E1 -21605.799,E2 -21605.799} C_VEL
LIN {X 0,Y 348.138,Z 600.092,A -85,B 0,C 180,E1 -21608.096,E2 -21608.096} C_VEL
LIN {X 0,Y 350.28,Z 598.274,A -85,B 0,C 180,E1 -21610.368,E2 -21610.368} C_VEL
LIN {X 0,Y 353.114,Z 594.916,A -85,B 0,C 180,E1 -21612.603,E2 -21612.603} C_VEL
LIN {X 0,Y 356.122,Z 590.09,A -85,B 0,C 180,E1 -21614.814,E2 -21614.814} C_VEL
LIN {X 0,Y 358.629,Z 585.349,A -85,B 0,C 180,E1 -21616.451,E2 -21616.451} C_VEL
LIN {X 0,Y 361.866,Z 578.619,A -85,B 0,C 180,E1 -21618.303,E2 -21618.303} C_VEL
LIN {X 0,Y 365.412,Z 570.077,A -85,B 0,C 180,E1 -21620.184,E2 -21620.184} C_VEL
LIN {X 0,Y 368.688,Z 561.237,A -85,B 0,C 180,E1 -21621.744,E2 -21621.744} C_VEL
LIN {X 0,Y 372.207,Z 550.623,A -85,B 0,C 180,E1 -21623.278,E2 -21623.278} C_VEL
LIN {X 0,Y 375.637,Z 538.865,A -85,B 0,C 180,E1 -21624.659,E2 -21624.659} C_VEL
LIN {X 0,Y 378.868,Z 525.791,A -85,B 0,C 180,E1 -21625.898,E2 -21625.898} C_VEL
LIN {X 0,Y 381.709,Z 511.447,A -85,B 0,C 180,E1 -21627.011,E2 -21627.011} C_VEL
LIN {X 0,Y 384.105,Z 495.944,A -85,B 0,C 180,E1 -21627.932,E2 -21627.932} C_VEL
LIN {X 0,Y 385.954,Z 479.777,A -85,B 0,C 180,E1 -21628.635,E2 -21628.635} C_VEL
LIN {X 0,Y 389.189,Z 453.372,A -85,B 0,C 180,E1 -21629.559,E2 -21629.559} C_VEL
LIN {X 0,Y 393.603,Z 420.938,A -85,B 0,C 180,E1 -21630.649,E2 -21630.649} C_VEL
LIN {X 0,Y 390.526,Z 414.611,A -85,B 0,C 180,E1 -21631.96,E2 -21631.96} C_VEL
LIN {X 0,Y 387.144,Z 408.283,A -85,B 0,C 180,E1 -21633.584,E2 -21633.584} C_VEL
LIN {X 0,Y 384.407,Z 403.861,A -85,B 0,C 180,E1 -21635.091,E2 -21635.091} C_VEL
LIN {X 0,Y 382.331,Z 400.377,A -85,B 0,C 180,E1 -21636.494,E2 -21636.494} C_VEL
LIN {X 0,Y 380.257,Z 397.23,A -85,B 0,C 180,E1 -21638.209,E2 -21638.209} C_VEL
LIN {X 0,Y 379.649,Z 396.059,A -85,B 0,C 180,E1 -21638.85,E2 -21638.85} C_VEL
LIN {X 0,Y 377.608,Z 394.247,A -85,B 0,C 180,E1 -21641.896,E2 -21641.896} C_VEL
LIN {X 0,Y 377.382,Z 394.072,A -85,B 0,C 180,E1 -21644.245,E2 -21644.245} C_VEL
LIN {X 0,Y 378.56,Z 395.463,A -85,B 0,C 180,E1 -21646.963,E2 -21646.963} C_VEL
LIN {X 0,Y 379.636,Z 396.536,A -85,B 0,C 180,E1 -21648.159,E2 -21648.159} C_VEL
LIN {X 0,Y 381.312,Z 399.683,A -85,B 0,C 180,E1 -21649.836,E2 -21649.836} C_VEL
LIN {X 0,Y 382.478,Z 401.177,A -85,B 0,C 180,E1 -21650.691,E2 -21650.691} C_VEL
LIN {X 0,Y 383.831,Z 409.016,A -85,B 0,C 180,E1 -21652.217,E2 -21652.217} C_VEL
LIN {X 0,Y 386.188,Z 422.607,A -85,B 0,C 180,E1 -21654.343,E2 -21654.343} C_VEL
LIN {X 0,Y 386.369,Z 443.033,A -85,B 0,C 180,E1 -21656.026,E2 -21656.026} C_VEL
LIN {X 0,Y 386.38,Z 463.13,A -85,B 0,C 180,E1 -21657.457,E2 -21657.457} C_VEL
LIN {X 0,Y 386.206,Z 476.293,A -85,B 0,C 180,E1 -21658.267,E2 -21658.267} C_VEL
LIN {X 0,Y 385.385,Z 490.635,A -85,B 0,C 180,E1 -21658.988,E2 -21658.988} C_VEL
LIN {X 0,Y 379.333,Z 538.183,A -85,B 0,C 180,E1 -21660.59,E2 -21660.59} C_VEL
LIN {X 0,Y 376.32,Z 554.291,A -85,B 0,C 180,E1 -21661.294,E2 -21661.294} C_VEL
LIN {X 0,Y 372.904,Z 569.204,A -85,B 0,C 180,E1 -21662.144,E2 -21662.144} C_VEL
LIN {X 0,Y 368.98,Z 583.679,A -85,B 0,C 180,E1 -21663.201,E2 -21663.201} C_VEL
LIN {X 0,Y 364.966,Z 596.858,A -85,B 0,C 180,E1 -21664.416,E2 -21664.416} C_VEL
LIN {X 0,Y 361.333,Z 608.023,A -85,B 0,C 180,E1 -21665.674,E2 -21665.674} C_VEL
LIN {X 0,Y 357.404,Z 619.404,A -85,B 0,C 180,E1 -21667.252,E2 -21667.252} C_VEL
LIN {X 0,Y 353.54,Z 630.251,A -85,B 0,C 180,E1 -21669.107,E2 -21669.107} C_VEL
LIN {X 0,Y 350.311,Z 639.398,A -85,B 0,C 180,E1 -21671.039,E2 -21671.039} C_VEL
LIN {X 0,Y 347.614,Z 646.929,A -85,B 0,C 180,E1 -21673.011,E2 -21673.011} C_VEL
LIN {X 0,Y 345.915,Z 652.309,A -85,B 0,C 180,E1 -21674.738,E2 -21674.738} C_VEL
LIN {X 0,Y 344.307,Z 658.1,A -85,B 0,C 180,E1 -21677.069,E2 -21677.069} C_VEL
LIN {X 0,Y 343.504,Z 662.214,A -85,B 0,C 180,E1 -21679.202,E2 -21679.202} C_VEL
LIN {X 0,Y 343.099,Z 671.703,A -85,B 0,C 180,E1 -21680.896,E2 -21680.896} C_VEL
LIN {X 0,Y 342.728,Z 681.14,A -85,B 0,C 180,E1 -21682.956,E2 -21682.956} C_VEL
LIN {X 0,Y 342.587,Z 687.738,A -85,B 0,C 180,E1 -21684.721,E2 -21684.721} C_VEL
LIN {X 0,Y 342.479,Z 693.108,A -85,B 0,C 180,E1 -21686.482,E2 -21686.482} C_VEL
LIN {X 0,Y 342.405,Z 697.384,A -85,B 0,C 180,E1 -21688.241,E2 -21688.241} C_VEL
LIN {X 0,Y 342.405,Z 700.723,A -85,B 0,C 180,E1 -21690,E2 -21690} C_VEL
LIN {X 0,Y 342.298,Z 703.772,A -85,B 0,C 180,E1 -21692.345,E2 -21692.345} C_VEL
LIN {X 0,Y 342.409,Z 705.368,A -85,B 0,C 180,E1 -21694.693,E2 -21694.693} C_VEL
LIN {X 0,Y 342.954,Z 705.554,A -85,B 0,C 180,E1 -21697.039,E2 -21697.039} C_VEL
LIN {X 0,Y 343.845,Z 704.352,A -85,B 0,C 180,E1 -21699.379,E2 -21699.379} C_VEL
LIN {X 0,Y 345.397,Z 701.757,A -85,B 0,C 180,E1 -21701.7,E2 -21701.7} C_VEL
LIN {X 0,Y 347.7,Z 697.672,A -85,B 0,C 180,E1 -21703.989,E2 -21703.989} C_VEL
LIN {X 0,Y 350.174,Z 692.084,A -85,B 0,C 180,E1 -21706.262,E2 -21706.262} C_VEL
LIN {X 0,Y 353.05,Z 685.799,A -85,B 0,C 180,E1 -21708.208,E2 -21708.208} C_VEL
LIN {X 0,Y 356.404,Z 678.058,A -85,B 0,C 180,E1 -21710.116,E2 -21710.116} C_VEL
LIN {X 0,Y 360.16,Z 668.644,A -85,B 0,C 180,E1 -21711.986,E2 -21711.986} C_VEL
LIN {X 0,Y 363.785,Z 658.938,A -85,B 0,C 180,E1 -21713.549,E2 -21713.549} C_VEL
LIN {X 0,Y 367.727,Z 647.33,A -85,B 0,C 180,E1 -21715.076,E2 -21715.076} C_VEL
LIN {X 0,Y 372.022,Z 633.264,A -85,B 0,C 180,E1 -21716.562,E2 -21716.562} C_VEL
LIN {X 0,Y 375.598,Z 620.246,A -85,B 0,C 180,E1 -21717.638,E2 -21717.638} C_VEL
LIN {X 0,Y 378.537,Z 607.998,A -85,B 0,C 180,E1 -21718.456,E2 -21718.456} C_VEL
LIN {X 0,Y 381.713,Z 592.598,A -85,B 0,C 180,E1 -21719.247,E2 -21719.247} C_VEL
LIN {X 0,Y 384.445,Z 574.971,A -85,B 0,C 180,E1 -21719.918,E2 -21719.918} C_VEL
LIN {X 0,Y 396.312,Z 492.244,A -85,B 0,C 180,E1 -21722.719,E2 -21722.719} C_VEL
LIN {X 0,Y 397.058,Z 481.341,A -85,B 0,C 180,E1 -21723.34,E2 -21723.34} C_VEL
LIN {X 0,Y 397.718,Z 466.667,A -85,B 0,C 180,E1 -21724.328,E2 -21724.328} C_VEL
LIN {X 0,Y 398.051,Z 450.689,A -85,B 0,C 180,E1 -21725.645,E2 -21725.645} C_VEL
LIN {X 0,Y 398.125,Z 439.836,A -85,B 0,C 180,E1 -21726.718,E2 -21726.718} C_VEL
LIN {X 0,Y 396.951,Z 438.327,A -85,B 0,C 180,E1 -21727.434,E2 -21727.434} C_VEL
LIN {X 0,Y 394.677,Z 435.329,A -85,B 0,C 180,E1 -21729.71,E2 -21729.71} C_VEL
LIN {X 0,Y 393.282,Z 434.09,A -85,B 0,C 180,E1 -21731.58,E2 -21731.58} C_VEL
LIN {X 0,Y 392.539,Z 433.796,A -85,B 0,C 180,E1 -21732.979,E2 -21732.979} C_VEL
LIN {X 0,Y 391.989,Z 434.015,A -85,B 0,C 180,E1 -21734.377,E2 -21734.377} C_VEL
LIN {X 0,Y 391.588,Z 434.782,A -85,B 0,C 180,E1 -21735.765,E2 -21735.765} C_VEL
LIN {X 0,Y 391.322,Z 436.265,A -85,B 0,C 180,E1 -21737.212,E2 -21737.212} C_VEL
LIN {X 0,Y 391.234,Z 439.594,A -85,B 0,C 180,E1 -21739.404,E2 -21739.404} C_VEL
LIN {X 0,Y 393.143,Z 445.778,A -85,B 0,C 180,E1 -21741.622,E2 -21741.622} C_VEL
LIN {X 0,Y 394.964,Z 452.219,A -85,B 0,C 180,E1 -21743.234,E2 -21743.234} C_VEL
LIN {X 0,Y 395.398,Z 468.817,A -85,B 0,C 180,E1 -21745.019,E2 -21745.019} C_VEL
LIN {X 0,Y 395.764,Z 482.268,A -85,B 0,C 180,E1 -21746.266,E2 -21746.266} C_VEL
LIN {X 0,Y 395.943,Z 495.512,A -85,B 0,C 180,E1 -21747.326,E2 -21747.326} C_VEL
LIN {X 0,Y 395.549,Z 498.976,A -85,B 0,C 180,E1 -21747.476,E2 -21747.476} C_VEL
LIN {X 0,Y 383.244,Z 585.188,A -85,B 0,C 180,E1 -21750.394,E2 -21750.394} C_VEL
LIN {X 0,Y 380.374,Z 600.299,A -85,B 0,C 180,E1 -21751.094,E2 -21751.094} C_VEL
LIN {X 0,Y 377.381,Z 613.548,A -85,B 0,C 180,E1 -21751.903,E2 -21751.903} C_VEL
LIN {X 0,Y 373.819,Z 627.401,A -85,B 0,C 180,E1 -21752.975,E2 -21752.975} C_VEL
LIN {X 0,Y 370.429,Z 638.857,A -85,B 0,C 180,E1 -21754.07,E2 -21754.07} C_VEL
LIN {X 0,Y 366.646,Z 650.629,A -85,B 0,C 180,E1 -21755.448,E2 -21755.448} C_VEL
LIN {X 0,Y 362.794,Z 661.428,A -85,B 0,C 180,E1 -21756.986,E2 -21756.986} C_VEL
LIN {X 0,Y 358.748,Z 671.88,A -85,B 0,C 180,E1 -21758.826,E2 -21758.826} C_VEL
LIN {X 0,Y 355.696,Z 679.352,A -85,B 0,C 180,E1 -21760.442,E2 -21760.442} C_VEL
LIN {X 0,Y 352.06,Z 687.475,A -85,B 0,C 180,E1 -21762.637,E2 -21762.637} C_VEL
LIN {X 0,Y 349.731,Z 692.42,A -85,B 0,C 180,E1 -21764.313,E2 -21764.313} C_VEL
LIN {X 0,Y 347.954,Z 696.406,A -85,B 0,C 180,E1 -21766.021,E2 -21766.021} C_VEL
LIN {X 0,Y 345.618,Z 700.46,A -85,B 0,C 180,E1 -21768.307,E2 -21768.307} C_VEL
LIN {X 0,Y 344.01,Z 703.036,A -85,B 0,C 180,E1 -21770.626,E2 -21770.626} C_VEL
LIN {X 0,Y 342.999,Z 704.219,A -85,B 0,C 180,E1 -21772.962,E2 -21772.962} C_VEL
LIN {X 0,Y 342.41,Z 704.022,A -85,B 0,C 180,E1 -21775.307,E2 -21775.307} C_VEL
LIN {X 0,Y 342.201,Z 702.425,A -85,B 0,C 180,E1 -21777.654,E2 -21777.654} C_VEL
LIN {X 0,Y 342.293,Z 699.396,A -85,B 0,C 180,E1 -21780,E2 -21780} C_VEL
LIN {X 0,Y 342.333,Z 696.096,A -85,B 0,C 180,E1 -21781.759,E2 -21781.759} C_VEL
LIN {X 0,Y 342.389,Z 691.862,A -85,B 0,C 180,E1 -21783.519,E2 -21783.519} C_VEL
LIN {X 0,Y 342.554,Z 685.562,A -85,B 0,C 180,E1 -21785.574,E2 -21785.574} C_VEL
LIN {X 0,Y 342.815,Z 677.61,A -85,B 0,C 180,E1 -21787.632,E2 -21787.632} C_VEL
LIN {X 0,Y 343.219,Z 669.302,A -85,B 0,C 180,E1 -21789.397,E2 -21789.397} C_VEL
LIN {X 0,Y 343.739,Z 659.294,A -85,B 0,C 180,E1 -21791.162,E2 -21791.162} C_VEL
LIN {X 0,Y 344.511,Z 648.662,A -85,B 0,C 180,E1 -21792.726,E2 -21792.726} C_VEL
LIN {X 0,Y 345.226,Z 636.127,A -85,B 0,C 180,E1 -21794.242,E2 -21794.242} C_VEL
LIN {X 0,Y 346.118,Z 622.781,A -85,B 0,C 180,E1 -21795.554,E2 -21795.554} C_VEL
LIN {X 0,Y 346.945,Z 608.997,A -85,B 0,C 180,E1 -21796.645,E2 -21796.645} C_VEL
LIN {X 0,Y 347.71,Z 594.134,A -85,B 0,C 180,E1 -21797.55,E2 -21797.55} C_VEL
LIN {X 0,Y 348.323,Z 578.691,A -85,B 0,C 180,E1 -21798.237,E2 -21798.237} C_VEL
LIN {X 0,Y 351.714,Z 475.894,A -85,B 0,C 180,E1 -21801.504,E2 -21801.504} C_VEL
LIN {X 0,Y 349.273,Z 446.356,A -85,B 0,C 180,E1 -21802.519,E2 -21802.519} C_VEL
LIN {X 0,Y 349.021,Z 439.487,A -85,B 0,C 180,E1 -21802.771,E2 -21802.771} C_VEL
LIN {X 0,Y 351.217,Z 413.209,A -85,B 0,C 180,E1 -21806.598,E2 -21806.598} C_VEL
LIN {X 0,Y 353.022,Z 391.681,A -85,B 0,C 180,E1 -21809.738,E2 -21809.738} C_VEL
LIN {X 0,Y 348.806,Z 372.409,A -85,B 0,C 180,E1 -21812.833,E2 -21812.833} C_VEL
LIN {X 0,Y 344.93,Z 355.078,A -85,B 0,C 180,E1 -21815.705,E2 -21815.705} C_VEL
LIN {X 0,Y 344.819,Z 355.088,A -85,B 0,C 180,E1 -21819.474,E2 -21819.474} C_VEL
LIN {X 0,Y 344.858,Z 355.088,A -85,B 0,C 180,E1 -21823.013,E2 -21823.013} C_VEL
LIN {X 0,Y 344.864,Z 355.08,A -85,B 0,C 180,E1 -21826.325,E2 -21826.325} C_VEL
LIN {X 0,Y 344.817,Z 355.084,A -85,B 0,C 180,E1 -21829.456,E2 -21829.456} C_VEL
LIN {X 0,Y 344.853,Z 355.087,A -85,B 0,C 180,E1 -21832.458,E2 -21832.458} C_VEL
LIN {X 0,Y 344.843,Z 355.085,A -85,B 0,C 180,E1 -21835.338,E2 -21835.338} C_VEL
LIN {X 0,Y 344.871,Z 355.071,A -85,B 0,C 180,E1 -21838.544,E2 -21838.544} C_VEL
LIN {X 0,Y 344.897,Z 355.08,A -85,B 0,C 180,E1 -21842.154,E2 -21842.154} C_VEL
LIN {X 0,Y 344.895,Z 355.082,A -85,B 0,C 180,E1 -21846.051,E2 -21846.051} C_VEL
LIN {X 0,Y 344.893,Z 355.083,A -85,B 0,C 180,E1 -21848.672,E2 -21848.672} C_VEL
LIN {X 0,Y 346.035,Z 358.12,A -85,B 0,C 180,E1 -21848.833,E2 -21848.833} C_VEL
LIN {X 0,Y 354.883,Z 377.763,A -85,B 0,C 180,E1 -21849.917,E2 -21849.917} C_VEL
LIN {X 0,Y 359.06,Z 387.974,A -85,B 0,C 180,E1 -21850.428,E2 -21850.428} C_VEL
LIN {X 0,Y 357.58,Z 460.939,A -85,B 0,C 180,E1 -21851.883,E2 -21851.883} C_VEL
LIN {X 0,Y 357.37,Z 478.01,A -85,B 0,C 180,E1 -21852.314,E2 -21852.314} C_VEL
LIN {X 0,Y 356.857,Z 491.713,A -85,B 0,C 180,E1 -21852.877,E2 -21852.877} C_VEL
LIN {X 0,Y 355.991,Z 505.111,A -85,B 0,C 180,E1 -21853.644,E2 -21853.644} C_VEL
LIN {X 0,Y 354.976,Z 517.215,A -85,B 0,C 180,E1 -21854.551,E2 -21854.551} C_VEL
LIN {X 0,Y 353.863,Z 529.13,A -85,B 0,C 180,E1 -21855.675,E2 -21855.675} C_VEL
LIN {X 0,Y 352.503,Z 540.946,A -85,B 0,C 180,E1 -21857.049,E2 -21857.049} C_VEL
LIN {X 0,Y 350.999,Z 551.161,A -85,B 0,C 180,E1 -21858.489,E2 -21858.489} C_VEL
LIN {X 0,Y 349.464,Z 561.061,A -85,B 0,C 180,E1 -21860.191,E2 -21860.191} C_VEL
LIN {X 0,Y 348.152,Z 569.286,A -85,B 0,C 180,E1 -21861.904,E2 -21861.904} C_VEL
LIN {X 0,Y 347.065,Z 576.149,A -85,B 0,C 180,E1 -21863.627,E2 -21863.627} C_VEL
LIN {X 0,Y 346.074,Z 581.832,A -85,B 0,C 180,E1 -21865.356,E2 -21865.356} C_VEL
LIN {X 0,Y 345.145,Z 587.903,A -85,B 0,C 180,E1 -21867.674,E2 -21867.674} C_VEL
LIN {X 0,Y 344.606,Z 592.35,A -85,B 0,C 180,E1 -21870,E2 -21870} C_VEL
LIN {X 0,Y 344.212,Z 595.4,A -85,B 0,C 180,E1 -21872.333,E2 -21872.333} C_VEL
LIN {X 0,Y 344.232,Z 597.109,A -85,B 0,C 180,E1 -21874.669,E2 -21874.669} C_VEL
LIN {X 0,Y 344.403,Z 597.54,A -85,B 0,C 180,E1 -21877.009,E2 -21877.009} C_VEL
LIN {X 0,Y 344.886,Z 596.675,A -85,B 0,C 180,E1 -21879.351,E2 -21879.351} C_VEL
LIN {X 0,Y 345.582,Z 594.504,A -85,B 0,C 180,E1 -21881.694,E2 -21881.694} C_VEL
LIN {X 0,Y 346.812,Z 590.929,A -85,B 0,C 180,E1 -21884.026,E2 -21884.026} C_VEL
LIN {X 0,Y 348.336,Z 585.861,A -85,B 0,C 180,E1 -21886.351,E2 -21886.351} C_VEL
LIN {X 0,Y 349.686,Z 580.918,A -85,B 0,C 180,E1 -21888.088,E2 -21888.088} C_VEL
LIN {X 0,Y 351.666,Z 573.465,A -85,B 0,C 180,E1 -21890.196,E2 -21890.196} C_VEL
LIN {X 0,Y 353.662,Z 565.024,A -85,B 0,C 180,E1 -21892.105,E2 -21892.105} C_VEL
LIN {X 0,Y 355.745,Z 555.728,A -85,B 0,C 180,E1 -21893.806,E2 -21893.806} C_VEL
LIN {X 0,Y 357.809,Z 545.394,A -85,B 0,C 180,E1 -21895.355,E2 -21895.355} C_VEL
LIN {X 0,Y 359.811,Z 533.949,A -85,B 0,C 180,E1 -21896.755,E2 -21896.755} C_VEL
LIN {X 0,Y 361.541,Z 522.776,A -85,B 0,C 180,E1 -21897.866,E2 -21897.866} C_VEL
LIN {X 0,Y 362.914,Z 510.673,A -85,B 0,C 180,E1 -21898.85,E2 -21898.85} C_VEL
LIN {X 0,Y 364.066,Z 497.272,A -85,B 0,C 180,E1 -21899.698,E2 -21899.698} C_VEL
LIN {X 0,Y 364.915,Z 483.448,A -85,B 0,C 180,E1 -21900.335,E2 -21900.335} C_VEL
LIN {X 0,Y 365.295,Z 469.064,A -85,B 0,C 180,E1 -21900.779,E2 -21900.779} C_VEL
LIN {X 0,Y 367.344,Z 399.205,A -85,B 0,C 180,E1 -21902.144,E2 -21902.144} C_VEL
LIN {X 0,Y 358.613,Z 380.789,A -85,B 0,C 180,E1 -21903.375,E2 -21903.375} C_VEL
LIN {X 0,Y 348.054,Z 361.676,A -85,B 0,C 180,E1 -21904.896,E2 -21904.896} C_VEL
LIN {X 0,Y 345.12,Z 356.422,A -85,B 0,C 180,E1 -21905.339,E2 -21905.339} C_VEL
LIN {X 0,Y 344.833,Z 355.089,A -85,B 0,C 180,E1 -21905.438,E2 -21905.438} C_VEL
LIN {X 0,Y 344.81,Z 355.093,A -85,B 0,C 180,E1 -21909.031,E2 -21909.031} C_VEL
LIN {X 0,Y 344.8,Z 355.092,A -85,B 0,C 180,E1 -21912.097,E2 -21912.097} C_VEL
LIN {X 0,Y 344.802,Z 355.089,A -85,B 0,C 180,E1 -21915.317,E2 -21915.317} C_VEL
LIN {X 0,Y 344.827,Z 355.087,A -85,B 0,C 180,E1 -21918.728,E2 -21918.728} C_VEL
LIN {X 0,Y 344.784,Z 355.059,A -85,B 0,C 180,E1 -21921.998,E2 -21921.998} C_VEL
LIN {X 0,Y 344.138,Z 355.132,A -85,B 0,C 180,E1 -21922.972,E2 -21922.972} C_VEL
LIN {X 0,Y 341.281,Z 355.494,A -85,B 0,C 180,E1 -21924.557,E2 -21924.557} C_VEL
LIN {X 0,Y 338.854,Z 355.819,A -85,B 0,C 180,E1 -21925.84,E2 -21925.84} C_VEL
LIN {X 0,Y 337.822,Z 355.958,A -85,B 0,C 180,E1 -21926.833,E2 -21926.833} C_VEL
LIN {X 0,Y 337.745,Z 355.966,A -85,B 0,C 180,E1 -21927.169,E2 -21927.169} C_VEL
LIN {X 0,Y 337.789,Z 355.96,A -85,B 0,C 180,E1 -21930.566,E2 -21930.566} C_VEL
LIN {X 0,Y 337.821,Z 355.948,A -85,B 0,C 180,E1 -21934.188,E2 -21934.188} C_VEL
LIN {X 0,Y 337.879,Z 355.956,A -85,B 0,C 180,E1 -21937.258,E2 -21937.258} C_VEL
LIN {X 0,Y 344.007,Z 379.557,A -85,B 0,C 180,E1 -21938.192,E2 -21938.192} C_VEL
LIN {X 0,Y 341.445,Z 472.965,A -85,B 0,C 180,E1 -21941.188,E2 -21941.188} C_VEL
LIN {X 0,Y 341.075,Z 488.133,A -85,B 0,C 180,E1 -21941.903,E2 -21941.903} C_VEL
LIN {X 0,Y 340.469,Z 503.429,A -85,B 0,C 180,E1 -21942.875,E2 -21942.875} C_VEL
LIN {X 0,Y 339.809,Z 517.116,A -85,B 0,C 180,E1 -21943.996,E2 -21943.996} C_VEL
LIN {X 0,Y 339.047,Z 530.41,A -85,B 0,C 180,E1 -21945.34,E2 -21945.34} C_VEL
LIN {X 0,Y 338.371,Z 542.589,A -85,B 0,C 180,E1 -21946.838,E2 -21946.838} C_VEL
LIN {X 0,Y 337.956,Z 550.88,A -85,B 0,C 180,E1 -21948.038,E2 -21948.038} C_VEL
LIN {X 0,Y 337.366,Z 561.509,A -85,B 0,C 180,E1 -21949.835,E2 -21949.835} C_VEL
LIN {X 0,Y 336.953,Z 570.354,A -85,B 0,C 180,E1 -21951.633,E2 -21951.633} C_VEL
LIN {X 0,Y 336.643,Z 578.855,A -85,B 0,C 180,E1 -21953.728,E2 -21953.728} C_VEL
LIN {X 0,Y 336.645,Z 585.776,A -85,B 0,C 180,E1 -21955.824,E2 -21955.824} C_VEL
LIN {X 0,Y 336.684,Z 590.571,A -85,B 0,C 180,E1 -21957.615,E2 -21957.615} C_VEL
LIN {X 0,Y 337.016,Z 595.523,A -85,B 0,C 180,E1 -21960,E2 -21960} C_VEL
LIN {X 0,Y 337.715,Z 598.961,A -85,B 0,C 180,E1 -21962.377,E2 -21962.377} C_VEL
LIN {X 0,Y 338.906,Z 600.914,A -85,B 0,C 180,E1 -21964.742,E2 -21964.742} C_VEL
LIN {X 0,Y 340.372,Z 601.484,A -85,B 0,C 180,E1 -21967.092,E2 -21967.092} C_VEL
LIN {X 0,Y 342.217,Z 600.674,A -85,B 0,C 180,E1 -21969.424,E2 -21969.424} C_VEL
LIN {X 0,Y 344.844,Z 598.394,A -85,B 0,C 180,E1 -21971.719,E2 -21971.719} C_VEL
LIN {X 0,Y 347.958,Z 594.593,A -85,B 0,C 180,E1 -21973.978,E2 -21973.978} C_VEL
LIN {X 0,Y 351.251,Z 589.26,A -85,B 0,C 180,E1 -21976.211,E2 -21976.211} C_VEL
LIN {X 0,Y 355.074,Z 582.191,A -85,B 0,C 180,E1 -21978.398,E2 -21978.398} C_VEL
LIN {X 0,Y 358.674,Z 574.358,A -85,B 0,C 180,E1 -21980.281,E2 -21980.281} C_VEL
LIN {X 0,Y 362.612,Z 564.724,A -85,B 0,C 180,E1 -21982.128,E2 -21982.128} C_VEL
LIN {X 0,Y 366.324,Z 554.65,A -85,B 0,C 180,E1 -21983.674,E2 -21983.674} C_VEL
LIN {X 0,Y 369.844,Z 543.542,A -85,B 0,C 180,E1 -21985.072,E2 -21985.072} C_VEL
LIN {X 0,Y 373.608,Z 530.058,A -85,B 0,C 180,E1 -21986.44,E2 -21986.44} C_VEL
LIN {X 0,Y 376.605,Z 516.48,A -85,B 0,C 180,E1 -21987.558,E2 -21987.558} C_VEL
LIN {X 0,Y 379.271,Z 501.223,A -85,B 0,C 180,E1 -21988.546,E2 -21988.546} C_VEL
LIN {X 0,Y 381.329,Z 486.055,A -85,B 0,C 180,E1 -21989.279,E2 -21989.279} C_VEL
LIN {X 0,Y 384.071,Z 463.775,A -85,B 0,C 180,E1 -21990.105,E2 -21990.105} C_VEL
LIN {X 0,Y 389.645,Z 424.648,A -85,B 0,C 180,E1 -21991.445,E2 -21991.445} C_VEL
LIN {X 0,Y 386.184,Z 417.621,A -85,B 0,C 180,E1 -21993.067,E2 -21993.067} C_VEL
LIN {X 0,Y 383.708,Z 413.224,A -85,B 0,C 180,E1 -21994.373,E2 -21994.373} C_VEL
LIN {X 0,Y 382.02,Z 410.219,A -85,B 0,C 180,E1 -21995.402,E2 -21995.402} C_VEL
LIN {X 0,Y 380.161,Z 406.927,A -85,B 0,C 180,E1 -21996.747,E2 -21996.747} C_VEL
LIN {X 0,Y 378.156,Z 403.593,A -85,B 0,C 180,E1 -21998.569,E2 -21998.569} C_VEL
LIN {X 0,Y 377.699,Z 402.806,A -85,B 0,C 180,E1 -21999.089,E2 -21999.089} C_VEL
LIN {X 0,Y 375.815,Z 401.039,A -85,B 0,C 180,E1 -22002.142,E2 -22002.142} C_VEL
LIN {X 0,Y 375.736,Z 401.042,A -85,B 0,C 180,E1 -22004.49,E2 -22004.49} C_VEL
LIN {X 0,Y 377.029,Z 402.528,A -85,B 0,C 180,E1 -22007.212,E2 -22007.212} C_VEL
LIN {X 0,Y 377.723,Z 403.3,A -85,B 0,C 180,E1 -22007.979,E2 -22007.979} C_VEL
LIN {X 0,Y 379.276,Z 406.3,A -85,B 0,C 180,E1 -22009.615,E2 -22009.615} C_VEL
LIN {X 0,Y 380.146,Z 407.518,A -85,B 0,C 180,E1 -22010.302,E2 -22010.302} C_VEL
LIN {X 0,Y 381.141,Z 414.306,A -85,B 0,C 180,E1 -22011.631,E2 -22011.631} C_VEL
LIN {X 0,Y 382.917,Z 426.528,A -85,B 0,C 180,E1 -22013.597,E2 -22013.597} C_VEL
LIN {X 0,Y 382.743,Z 446.662,A -85,B 0,C 180,E1 -22015.28,E2 -22015.28} C_VEL
LIN {X 0,Y 382.501,Z 466.66,A -85,B 0,C 180,E1 -22016.722,E2 -22016.722} C_VEL
LIN {X 0,Y 382.077,Z 479.47,A -85,B 0,C 180,E1 -22017.517,E2 -22017.517} C_VEL
LIN {X 0,Y 381.218,Z 492.403,A -85,B 0,C 180,E1 -22018.16,E2 -22018.16} C_VEL
LIN {X 0,Y 374.915,Z 538.299,A -85,B 0,C 180,E1 -22019.745,E2 -22019.745} C_VEL
LIN {X 0,Y 371.827,Z 553.964,A -85,B 0,C 180,E1 -22020.441,E2 -22020.441} C_VEL
LIN {X 0,Y 368.219,Z 568.572,A -85,B 0,C 180,E1 -22021.293,E2 -22021.293} C_VEL
LIN {X 0,Y 363.692,Z 584.288,A -85,B 0,C 180,E1 -22022.469,E2 -22022.469} C_VEL
LIN {X 0,Y 359.117,Z 598.305,A -85,B 0,C 180,E1 -22023.813,E2 -22023.813} C_VEL
LIN {X 0,Y 355.011,Z 609.952,A -85,B 0,C 180,E1 -22025.212,E2 -22025.212} C_VEL
LIN {X 0,Y 351.001,Z 620.782,A -85,B 0,C 180,E1 -22026.796,E2 -22026.796} C_VEL
LIN {X 0,Y 346.987,Z 631.224,A -85,B 0,C 180,E1 -22028.693,E2 -22028.693} C_VEL
LIN {X 0,Y 343.157,Z 641.066,A -85,B 0,C 180,E1 -22030.938,E2 -22030.938} C_VEL
LIN {X 0,Y 340.829,Z 647.176,A -85,B 0,C 180,E1 -22032.663,E2 -22032.663} C_VEL
LIN {X 0,Y 338.53,Z 653.836,A -85,B 0,C 180,E1 -22035.011,E2 -22035.011} C_VEL
LIN {X 0,Y 337.357,Z 657.829,A -85,B 0,C 180,E1 -22036.797,E2 -22036.797} C_VEL
LIN {X 0,Y 336.419,Z 661.881,A -85,B 0,C 180,E1 -22039.2,E2 -22039.2} C_VEL
LIN {X 0,Y 336.408,Z 662.4,A -85,B 0,C 180,E1 -22039.351,E2 -22039.351} C_VEL
LIN {X 0,Y 336.017,Z 671.464,A -85,B 0,C 180,E1 -22041.005,E2 -22041.005} C_VEL
LIN {X 0,Y 335.663,Z 680.931,A -85,B 0,C 180,E1 -22043.108,E2 -22043.108} C_VEL
LIN {X 0,Y 335.515,Z 688.493,A -85,B 0,C 180,E1 -22045.21,E2 -22045.21} C_VEL
LIN {X 0,Y 335.397,Z 693.723,A -85,B 0,C 180,E1 -22047.007,E2 -22047.007} C_VEL
LIN {X 0,Y 335.345,Z 697.883,A -85,B 0,C 180,E1 -22048.803,E2 -22048.803} C_VEL
LIN {X 0,Y 335.329,Z 700.124,A -85,B 0,C 180,E1 -22050,E2 -22050} C_VEL
LIN {X 0,Y 335.224,Z 703.388,A -85,B 0,C 180,E1 -22052.395,E2 -22052.395} C_VEL
LIN {X 0,Y 335.346,Z 705.187,A -85,B 0,C 180,E1 -22054.792,E2 -22054.792} C_VEL
LIN {X 0,Y 335.901,Z 705.591,A -85,B 0,C 180,E1 -22057.187,E2 -22057.187} C_VEL
LIN {X 0,Y 336.839,Z 704.616,A -85,B 0,C 180,E1 -22059.576,E2 -22059.576} C_VEL
LIN {X 0,Y 338.474,Z 702.262,A -85,B 0,C 180,E1 -22061.943,E2 -22061.943} C_VEL
LIN {X 0,Y 340.871,Z 698.467,A -85,B 0,C 180,E1 -22064.275,E2 -22064.275} C_VEL
LIN {X 0,Y 343.456,Z 693.223,A -85,B 0,C 180,E1 -22066.59,E2 -22066.59} C_VEL
LIN {X 0,Y 346.924,Z 686.263,A -85,B 0,C 180,E1 -22068.847,E2 -22068.847} C_VEL
LIN {X 0,Y 350.463,Z 678.651,A -85,B 0,C 180,E1 -22070.778,E2 -22070.778} C_VEL
LIN {X 0,Y 354.412,Z 669.396,A -85,B 0,C 180,E1 -22072.668,E2 -22072.668} C_VEL
LIN {X 0,Y 358.222,Z 659.898,A -85,B 0,C 180,E1 -22074.244,E2 -22074.244} C_VEL
LIN {X 0,Y 362.72,Z 647.535,A -85,B 0,C 180,E1 -22075.907,E2 -22075.907} C_VEL
LIN {X 0,Y 366.846,Z 634.845,A -85,B 0,C 180,E1 -22077.274,E2 -22077.274} C_VEL
LIN {X 0,Y 370.579,Z 622.314,A -85,B 0,C 180,E1 -22078.353,E2 -22078.353} C_VEL
LIN {X 0,Y 374.074,Z 608.737,A -85,B 0,C 180,E1 -22079.287,E2 -22079.287} C_VEL
LIN {X 0,Y 377.361,Z 593.722,A -85,B 0,C 180,E1 -22080.077,E2 -22080.077} C_VEL
LIN {X 0,Y 380.235,Z 576.727,A -85,B 0,C 180,E1 -22080.743,E2 -22080.743} C_VEL
LIN {X 0,Y 392.842,Z 493.388,A -85,B 0,C 180,E1 -22083.602,E2 -22083.602} C_VEL
LIN {X 0,Y 393.925,Z 479.308,A -85,B 0,C 180,E1 -22084.452,E2 -22084.452} C_VEL
LIN {X 0,Y 394.539,Z 467.403,A -85,B 0,C 180,E1 -22085.314,E2 -22085.314} C_VEL
LIN {X 0,Y 395.082,Z 454.256,A -85,B 0,C 180,E1 -22086.419,E2 -22086.419} C_VEL
LIN {X 0,Y 395.324,Z 445.746,A -85,B 0,C 180,E1 -22087.248,E2 -22087.248} C_VEL
LIN {X 0,Y 392.532,Z 442.603,A -85,B 0,C 180,E1 -22089.102,E2 -22089.102} C_VEL
LIN {X 0,Y 390.509,Z 440.765,A -85,B 0,C 180,E1 -22090.886,E2 -22090.886} C_VEL
LIN {X 0,Y 389.251,Z 440.009,A -85,B 0,C 180,E1 -22092.457,E2 -22092.457} C_VEL
LIN {X 0,Y 388.361,Z 440.206,A -85,B 0,C 180,E1 -22094.455,E2 -22094.455} C_VEL
LIN {X 0,Y 388.216,Z 441.702,A -85,B 0,C 180,E1 -22096.314,E2 -22096.314} C_VEL
LIN {X 0,Y 388.929,Z 445.1,A -85,B 0,C 180,E1 -22098.616,E2 -22098.616} C_VEL
LIN {X 0,Y 390.019,Z 449.217,A -85,B 0,C 180,E1 -22100.302,E2 -22100.302} C_VEL
LIN {X 0,Y 391.099,Z 453.037,A -85,B 0,C 180,E1 -22101.53,E2 -22101.53} C_VEL
LIN {X 0,Y 392.184,Z 457.341,A -85,B 0,C 180,E1 -22102.61,E2 -22102.61} C_VEL
LIN {X 0,Y 392.258,Z 472.555,A -85,B 0,C 180,E1 -22104.268,E2 -22104.268} C_VEL
LIN {X 0,Y 392.356,Z 485.209,A -85,B 0,C 180,E1 -22105.468,E2 -22105.468} C_VEL
LIN {X 0,Y 392.329,Z 497.071,A -85,B 0,C 180,E1 -22106.446,E2 -22106.446} C_VEL
LIN {X 0,Y 392.079,Z 499.683,A -85,B 0,C 180,E1 -22106.583,E2 -22106.583} C_VEL
LIN {X 0,Y 379.063,Z 585.799,A -85,B 0,C 180,E1 -22109.536,E2 -22109.536} C_VEL
LIN {X 0,Y 376.245,Z 600.054,A -85,B 0,C 180,E1 -22110.21,E2 -22110.21} C_VEL
LIN {X 0,Y 372.834,Z 614.183,A -85,B 0,C 180,E1 -22111.069,E2 -22111.069} C_VEL
LIN {X 0,Y 369.106,Z 627.81,A -85,B 0,C 180,E1 -22112.141,E2 -22112.141} C_VEL
LIN {X 0,Y 365.578,Z 639.135,A -85,B 0,C 180,E1 -22113.24,E2 -22113.24} C_VEL
LIN {X 0,Y 361.935,Z 649.837,A -85,B 0,C 180,E1 -22114.495,E2 -22114.495} C_VEL
LIN {X 0,Y 357.819,Z 660.716,A -85,B 0,C 180,E1 -22116.035,E2 -22116.035} C_VEL
LIN {X 0,Y 353.529,Z 671.265,A -85,B 0,C 180,E1 -22117.887,E2 -22117.887} C_VEL
LIN {X 0,Y 349.685,Z 679.922,A -85,B 0,C 180,E1 -22119.786,E2 -22119.786} C_VEL
LIN {X 0,Y 346.32,Z 687.02,A -85,B 0,C 180,E1 -22121.73,E2 -22121.73} C_VEL
LIN {X 0,Y 342.986,Z 693.472,A -85,B 0,C 180,E1 -22123.997,E2 -22123.997} C_VEL
LIN {X 0,Y 341.118,Z 697.248,A -85,B 0,C 180,E1 -22125.735,E2 -22125.735} C_VEL
LIN {X 0,Y 338.697,Z 701.007,A -85,B 0,C 180,E1 -22128.065,E2 -22128.065} C_VEL
LIN {X 0,Y 336.998,Z 703.334,A -85,B 0,C 180,E1 -22130.429,E2 -22130.429} C_VEL
LIN {X 0,Y 335.968,Z 704.291,A -85,B 0,C 180,E1 -22132.814,E2 -22132.814} C_VEL
LIN {X 0,Y 335.348,Z 703.878,A -85,B 0,C 180,E1 -22135.208,E2 -22135.208} C_VEL
LIN {X 0,Y 335.126,Z 702.078,A -85,B 0,C 180,E1 -22137.605,E2 -22137.605} C_VEL
LIN {X 0,Y 335.223,Z 698.835,A -85,B 0,C 180,E1 -22140,E2 -22140} C_VEL
LIN {X 0,Y 335.263,Z 695.334,A -85,B 0,C 180,E1 -22141.796,E2 -22141.796} C_VEL
LIN {X 0,Y 335.345,Z 690.887,A -85,B 0,C 180,E1 -22143.593,E2 -22143.593} C_VEL
LIN {X 0,Y 335.5,Z 684.334,A -85,B 0,C 180,E1 -22145.692,E2 -22145.692} C_VEL
LIN {X 0,Y 335.74,Z 677.412,A -85,B 0,C 180,E1 -22147.493,E2 -22147.493} C_VEL
LIN {X 0,Y 336.151,Z 669.09,A -85,B 0,C 180,E1 -22149.294,E2 -22149.294} C_VEL
LIN {X 0,Y 336.651,Z 659.039,A -85,B 0,C 180,E1 -22151.097,E2 -22151.097} C_VEL
LIN {X 0,Y 337.429,Z 648.495,A -85,B 0,C 180,E1 -22152.673,E2 -22152.673} C_VEL
LIN {X 0,Y 338.159,Z 635.743,A -85,B 0,C 180,E1 -22154.24,E2 -22154.24} C_VEL
LIN {X 0,Y 339.032,Z 622.362,A -85,B 0,C 180,E1 -22155.58,E2 -22155.58} C_VEL
LIN {X 0,Y 339.885,Z 608.561,A -85,B 0,C 180,E1 -22156.692,E2 -22156.692} C_VEL
LIN {X 0,Y 340.628,Z 594.334,A -85,B 0,C 180,E1 -22157.58,E2 -22157.58} C_VEL
LIN {X 0,Y 341.224,Z 579.056,A -85,B 0,C 180,E1 -22158.282,E2 -22158.282} C_VEL
LIN {X 0,Y 344.691,Z 476.224,A -85,B 0,C 180,E1 -22161.651,E2 -22161.651} C_VEL
LIN {X 0,Y 342.283,Z 447.205,A -85,B 0,C 180,E1 -22162.67,E2 -22162.67} C_VEL
LIN {X 0,Y 342,Z 439.617,A -85,B 0,C 180,E1 -22162.941,E2 -22162.941} C_VEL
LIN {X 0,Y 344.283,Z 412.725,A -85,B 0,C 180,E1 -22166.916,E2 -22166.916} C_VEL
LIN {X 0,Y 346.058,Z 392.895,A -85,B 0,C 180,E1 -22169.848,E2 -22169.848} C_VEL
LIN {X 0,Y 341.615,Z 372.66,A -85,B 0,C 180,E1 -22173.15,E2 -22173.15} C_VEL
LIN {X 0,Y 337.878,Z 355.956,A -85,B 0,C 180,E1 -22175.973,E2 -22175.973} C_VEL
LIN {X 0,Y 337.772,Z 355.963,A -85,B 0,C 180,E1 -22180.005,E2 -22180.005} C_VEL
LIN {X 0,Y 337.813,Z 355.962,A -85,B 0,C 180,E1 -22183.472,E2 -22183.472} C_VEL
LIN {X 0,Y 337.81,Z 355.962,A -85,B 0,C 180,E1 -22186.823,E2 -22186.823} C_VEL
LIN {X 0,Y 337.774,Z 355.961,A -85,B 0,C 180,E1 -22190.11,E2 -22190.11} C_VEL
LIN {X 0,Y 337.813,Z 355.957,A -85,B 0,C 180,E1 -22193.965,E2 -22193.965} C_VEL
LIN {X 0,Y 337.783,Z 355.955,A -85,B 0,C 180,E1 -22197.374,E2 -22197.374} C_VEL
LIN {X 0,Y 337.825,Z 355.962,A -85,B 0,C 180,E1 -22200.556,E2 -22200.556} C_VEL
LIN {X 0,Y 337.828,Z 355.961,A -85,B 0,C 180,E1 -22204.189,E2 -22204.189} C_VEL
LIN {X 0,Y 337.831,Z 355.962,A -85,B 0,C 180,E1 -22206.8,E2 -22206.8} C_VEL
LIN {X 0,Y 337.848,Z 355.961,A -85,B 0,C 180,E1 -22208.117,E2 -22208.117} C_VEL
LIN {X 0,Y 338.967,Z 358.992,A -85,B 0,C 180,E1 -22208.299,E2 -22208.299} C_VEL
LIN {X 0,Y 347.467,Z 377.421,A -85,B 0,C 180,E1 -22209.371,E2 -22209.371} C_VEL
LIN {X 0,Y 352.526,Z 389.859,A -85,B 0,C 180,E1 -22210.013,E2 -22210.013} C_VEL
LIN {X 0,Y 350.951,Z 464.568,A -85,B 0,C 180,E1 -22211.528,E2 -22211.528} C_VEL
LIN {X 0,Y 350.722,Z 479.492,A -85,B 0,C 180,E1 -22211.93,E2 -22211.93} C_VEL
LIN {X 0,Y 350.194,Z 493.677,A -85,B 0,C 180,E1 -22212.541,E2 -22212.541} C_VEL
LIN {X 0,Y 349.203,Z 507.722,A -85,B 0,C 180,E1 -22213.392,E2 -22213.392} C_VEL
LIN {X 0,Y 348.049,Z 520.25,A -85,B 0,C 180,E1 -22214.385,E2 -22214.385} C_VEL
LIN {X 0,Y 346.793,Z 532.989,A -85,B 0,C 180,E1 -22215.675,E2 -22215.675} C_VEL
LIN {X 0,Y 345.36,Z 544.476,A -85,B 0,C 180,E1 -22217.109,E2 -22217.109} C_VEL
LIN {X 0,Y 343.852,Z 554.028,A -85,B 0,C 180,E1 -22218.544,E2 -22218.544} C_VEL
LIN {X 0,Y 342.311,Z 563.578,A -85,B 0,C 180,E1 -22220.281,E2 -22220.281} C_VEL
LIN {X 0,Y 341.011,Z 571.5,A -85,B 0,C 180,E1 -22222.031,E2 -22222.031} C_VEL
LIN {X 0,Y 339.691,Z 579.105,A -85,B 0,C 180,E1 -22224.082,E2 -22224.082} C_VEL
LIN {X 0,Y 338.826,Z 584.417,A -85,B 0,C 180,E1 -22225.851,E2 -22225.851} C_VEL
LIN {X 0,Y 337.915,Z 590.018,A -85,B 0,C 180,E1 -22228.218,E2 -22228.218} C_VEL
LIN {X 0,Y 337.55,Z 593.206,A -85,B 0,C 180,E1 -22230,E2 -22230} C_VEL
LIN {X 0,Y 337.151,Z 596.224,A -85,B 0,C 180,E1 -22232.382,E2 -22232.382} C_VEL
LIN {X 0,Y 337.174,Z 597.902,A -85,B 0,C 180,E1 -22234.767,E2 -22234.767} C_VEL
LIN {X 0,Y 337.385,Z 598.299,A -85,B 0,C 180,E1 -22237.156,E2 -22237.156} C_VEL
LIN {X 0,Y 337.891,Z 597.405,A -85,B 0,C 180,E1 -22239.546,E2 -22239.546} C_VEL
LIN {X 0,Y 338.638,Z 595.201,A -85,B 0,C 180,E1 -22241.938,E2 -22241.938} C_VEL
LIN {X 0,Y 339.944,Z 591.591,A -85,B 0,C 180,E1 -22244.315,E2 -22244.315} C_VEL
LIN {X 0,Y 341.525,Z 586.481,A -85,B 0,C 180,E1 -22246.686,E2 -22246.686} C_VEL
LIN {X 0,Y 342.928,Z 581.508,A -85,B 0,C 180,E1 -22248.457,E2 -22248.457} C_VEL
LIN {X 0,Y 344.94,Z 574.196,A -85,B 0,C 180,E1 -22250.556,E2 -22250.556} C_VEL
LIN {X 0,Y 347.088,Z 565.498,A -85,B 0,C 180,E1 -22252.547,E2 -22252.547} C_VEL
LIN {X 0,Y 349.241,Z 556.139,A -85,B 0,C 180,E1 -22254.278,E2 -22254.278} C_VEL
LIN {X 0,Y 351.382,Z 545.733,A -85,B 0,C 180,E1 -22255.853,E2 -22255.853} C_VEL
LIN {X 0,Y 353.227,Z 535.482,A -85,B 0,C 180,E1 -22257.135,E2 -22257.135} C_VEL
LIN {X 0,Y 355.263,Z 522.904,A -85,B 0,C 180,E1 -22258.402,E2 -22258.402} C_VEL
LIN {X 0,Y 356.66,Z 510.634,A -85,B 0,C 180,E1 -22259.405,E2 -22259.405} C_VEL
LIN {X 0,Y 357.83,Z 497.555,A -85,B 0,C 180,E1 -22260.233,E2 -22260.233} C_VEL
LIN {X 0,Y 358.692,Z 483.638,A -85,B 0,C 180,E1 -22260.878,E2 -22260.878} C_VEL
LIN {X 0,Y 359.105,Z 468.88,A -85,B 0,C 180,E1 -22261.328,E2 -22261.328} C_VEL
LIN {X 0,Y 361.06,Z 400.903,A -85,B 0,C 180,E1 -22262.683,E2 -22262.683} C_VEL
LIN {X 0,Y 352.694,Z 383.581,A -85,B 0,C 180,E1 -22263.896,E2 -22263.896} C_VEL
LIN {X 0,Y 342.704,Z 365.392,A -85,B 0,C 180,E1 -22265.383,E2 -22265.383} C_VEL
LIN {X 0,Y 339.182,Z 359.411,A -85,B 0,C 180,E1 -22265.924,E2 -22265.924} C_VEL
LIN {X 0,Y 337.94,Z 356.828,A -85,B 0,C 180,E1 -22266.131,E2 -22266.131} C_VEL
LIN {X 0,Y 337.781,Z 355.966,A -85,B 0,C 180,E1 -22266.202,E2 -22266.202} C_VEL
LIN {X 0,Y 337.746,Z 355.971,A -85,B 0,C 180,E1 -22270.009,E2 -22270.009} C_VEL
LIN {X 0,Y 337.749,Z 355.975,A -85,B 0,C 180,E1 -22273.46,E2 -22273.46} C_VEL
LIN {X 0,Y 337.758,Z 355.971,A -85,B 0,C 180,E1 -22276.814,E2 -22276.814} C_VEL
LIN {X 0,Y 337.752,Z 355.968,A -85,B 0,C 180,E1 -22280.115,E2 -22280.115} C_VEL
LIN {X 0,Y 337.78,Z 355.923,A -85,B 0,C 180,E1 -22283.973,E2 -22283.973} C_VEL
LIN {X 0,Y 337.745,Z 355.966,A -85,B 0,C 180,E1 -22287.169,E2 -22287.169} C_VEL
LIN {X 0,Y 337.093,Z 356.057,A -85,B 0,C 180,E1 -22288.165,E2 -22288.165} C_VEL
LIN {X 0,Y 334.246,Z 356.415,A -85,B 0,C 180,E1 -22289.786,E2 -22289.786} C_VEL
LIN {X 0,Y 331.84,Z 356.709,A -85,B 0,C 180,E1 -22291.099,E2 -22291.099} C_VEL
LIN {X 0,Y 330.83,Z 356.831,A -85,B 0,C 180,E1 -22292.115,E2 -22292.115} C_VEL
LIN {X 0,Y 330.76,Z 356.837,A -85,B 0,C 180,E1 -22292.459,E2 -22292.459} C_VEL
LIN {X 0,Y 330.767,Z 356.841,A -85,B 0,C 180,E1 -22296.274,E2 -22296.274} C_VEL
LIN {X 0,Y 330.819,Z 356.835,A -85,B 0,C 180,E1 -22297.1,E2 -22297.1} C_VEL
LIN {X 0,Y 336.637,Z 379.185,A -85,B 0,C 180,E1 -22298.019,E2 -22298.019} C_VEL
LIN {X 0,Y 336.909,Z 381.9,A -85,B 0,C 180,E1 -22298.116,E2 -22298.116} C_VEL
LIN {X 0,Y 334.363,Z 473.366,A -85,B 0,C 180,E1 -22301.131,E2 -22301.131} C_VEL
LIN {X 0,Y 333.998,Z 487.837,A -85,B 0,C 180,E1 -22301.823,E2 -22301.823} C_VEL
LIN {X 0,Y 333.4,Z 503.353,A -85,B 0,C 180,E1 -22302.816,E2 -22302.816} C_VEL
LIN {X 0,Y 332.701,Z 517.169,A -85,B 0,C 180,E1 -22303.959,E2 -22303.959} C_VEL
LIN {X 0,Y 331.938,Z 530.599,A -85,B 0,C 180,E1 -22305.331,E2 -22305.331} C_VEL
LIN {X 0,Y 331.267,Z 542.925,A -85,B 0,C 180,E1 -22306.861,E2 -22306.861} C_VEL
LIN {X 0,Y 330.72,Z 553.193,A -85,B 0,C 180,E1 -22308.392,E2 -22308.392} C_VEL
LIN {X 0,Y 330.143,Z 563.512,A -85,B 0,C 180,E1 -22310.227,E2 -22310.227} C_VEL
LIN {X 0,Y 329.789,Z 572.18,A -85,B 0,C 180,E1 -22312.064,E2 -22312.064} C_VEL
LIN {X 0,Y 329.531,Z 580.558,A -85,B 0,C 180,E1 -22314.205,E2 -22314.205} C_VEL
LIN {X 0,Y 329.556,Z 587.331,A -85,B 0,C 180,E1 -22316.344,E2 -22316.344} C_VEL
LIN {X 0,Y 329.73,Z 593.351,A -85,B 0,C 180,E1 -22318.782,E2 -22318.782} C_VEL
LIN {X 0,Y 330.26,Z 597.779,A -85,B 0,C 180,E1 -22321.215,E2 -22321.215} C_VEL
LIN {X 0,Y 331.227,Z 600.744,A -85,B 0,C 180,E1 -22323.637,E2 -22323.637} C_VEL
LIN {X 0,Y 332.597,Z 602.295,A -85,B 0,C 180,E1 -22326.044,E2 -22326.044} C_VEL
LIN {X 0,Y 334.291,Z 602.428,A -85,B 0,C 180,E1 -22328.434,E2 -22328.434} C_VEL
LIN {X 0,Y 336.605,Z 601.144,A -85,B 0,C 180,E1 -22330.794,E2 -22330.794} C_VEL
LIN {X 0,Y 339.686,Z 598.369,A -85,B 0,C 180,E1 -22333.11,E2 -22333.11} C_VEL
LIN {X 0,Y 342.975,Z 594.172,A -85,B 0,C 180,E1 -22335.396,E2 -22335.396} C_VEL
LIN {X 0,Y 345.715,Z 589.945,A -85,B 0,C 180,E1 -22337.084,E2 -22337.084} C_VEL
LIN {X 0,Y 349.524,Z 583.294,A -85,B 0,C 180,E1 -22339.157,E2 -22339.157} C_VEL
LIN {X 0,Y 353.061,Z 576.153,A -85,B 0,C 180,E1 -22340.922,E2 -22340.922} C_VEL
LIN {X 0,Y 357.206,Z 566.689,A -85,B 0,C 180,E1 -22342.785,E2 -22342.785} C_VEL
LIN {X 0,Y 361.082,Z 556.825,A -85,B 0,C 180,E1 -22344.344,E2 -22344.344} C_VEL
LIN {X 0,Y 364.819,Z 546.1,A -85,B 0,C 180,E1 -22345.747,E2 -22345.747} C_VEL
LIN {X 0,Y 368.707,Z 532.925,A -85,B 0,C 180,E1 -22347.125,E2 -22347.125} C_VEL
LIN {X 0,Y 371.87,Z 519.949,A -85,B 0,C 180,E1 -22348.245,E2 -22348.245} C_VEL
LIN {X 0,Y 374.571,Z 506.477,A -85,B 0,C 180,E1 -22349.167,E2 -22349.167} C_VEL
LIN {X 0,Y 376.664,Z 492.875,A -85,B 0,C 180,E1 -22349.908,E2 -22349.908} C_VEL
LIN {X 0,Y 380.107,Z 466.527,A -85,B 0,C 180,E1 -22350.947,E2 -22350.947} C_VEL
LIN {X 0,Y 385.801,Z 428.634,A -85,B 0,C 180,E1 -22352.247,E2 -22352.247} C_VEL
LIN {X 0,Y 382.708,Z 422.196,A -85,B 0,C 180,E1 -22353.854,E2 -22353.854} C_VEL
LIN {X 0,Y 379.737,Z 416.695,A -85,B 0,C 180,E1 -22355.672,E2 -22355.672} C_VEL
LIN {X 0,Y 377.933,Z 413.413,A -85,B 0,C 180,E1 -22357.047,E2 -22357.047} C_VEL
LIN {X 0,Y 375.828,Z 409.617,A -85,B 0,C 180,E1 -22359.218,E2 -22359.218} C_VEL
LIN {X 0,Y 374.189,Z 408.024,A -85,B 0,C 180,E1 -22361.911,E2 -22361.911} C_VEL
LIN {X 0,Y 373.991,Z 407.826,A -85,B 0,C 180,E1 -22364.217,E2 -22364.217} C_VEL
LIN {X 0,Y 375.299,Z 409.409,A -85,B 0,C 180,E1 -22367.194,E2 -22367.194} C_VEL
LIN {X 0,Y 375.82,Z 410.136,A -85,B 0,C 180,E1 -22367.817,E2 -22367.817} C_VEL
LIN {X 0,Y 377.569,Z 413.331,A -85,B 0,C 180,E1 -22369.65,E2 -22369.65} C_VEL
LIN {X 0,Y 377.878,Z 414.008,A -85,B 0,C 180,E1 -22369.936,E2 -22369.936} C_VEL
LIN {X 0,Y 378.5,Z 419.464,A -85,B 0,C 180,E1 -22371.009,E2 -22371.009} C_VEL
LIN {X 0,Y 379.812,Z 430.803,A -85,B 0,C 180,E1 -22372.858,E2 -22372.858} C_VEL
LIN {X 0,Y 379.318,Z 449.508,A -85,B 0,C 180,E1 -22374.447,E2 -22374.447} C_VEL
LIN {X 0,Y 378.741,Z 469.315,A -85,B 0,C 180,E1 -22375.909,E2 -22375.909} C_VEL
LIN {X 0,Y 378.207,Z 481.621,A -85,B 0,C 180,E1 -22376.677,E2 -22376.677} C_VEL
LIN {X 0,Y 377.266,Z 493.359,A -85,B 0,C 180,E1 -22377.283,E2 -22377.283} C_VEL
LIN {X 0,Y 371.089,Z 536.177,A -85,B 0,C 180,E1 -22378.769,E2 -22378.769} C_VEL
LIN {X 0,Y 367.64,Z 552.813,A -85,B 0,C 180,E1 -22379.517,E2 -22379.517} C_VEL
LIN {X 0,Y 363.156,Z 569.933,A -85,B 0,C 180,E1 -22380.538,E2 -22380.538} C_VEL
LIN {X 0,Y 358.835,Z 584.024,A -85,B 0,C 180,E1 -22381.629,E2 -22381.629} C_VEL
LIN {X 0,Y 354.149,Z 597.466,A -85,B 0,C 180,E1 -22382.941,E2 -22382.941} C_VEL
LIN {X 0,Y 349.456,Z 610.066,A -85,B 0,C 180,E1 -22384.472,E2 -22384.472} C_VEL
LIN {X 0,Y 345.279,Z 620.555,A -85,B 0,C 180,E1 -22386.063,E2 -22386.063} C_VEL
LIN {X 0,Y 341.02,Z 630.831,A -85,B 0,C 180,E1 -22387.985,E2 -22387.985} C_VEL
LIN {X 0,Y 337.485,Z 639.403,A -85,B 0,C 180,E1 -22389.973,E2 -22389.973} C_VEL
LIN {X 0,Y 334.758,Z 645.575,A -85,B 0,C 180,E1 -22391.708,E2 -22391.708} C_VEL
LIN {X 0,Y 332.155,Z 652.332,A -85,B 0,C 180,E1 -22394.089,E2 -22394.089} C_VEL
LIN {X 0,Y 330.41,Z 657.549,A -85,B 0,C 180,E1 -22396.515,E2 -22396.515} C_VEL
LIN {X 0,Y 329.388,Z 661.376,A -85,B 0,C 180,E1 -22398.966,E2 -22398.966} C_VEL
LIN {X 0,Y 329.335,Z 662.036,A -85,B 0,C 180,E1 -22399.43,E2 -22399.43} C_VEL
LIN {X 0,Y 328.956,Z 671.143,A -85,B 0,C 180,E1 -22401.119,E2 -22401.119} C_VEL
LIN {X 0,Y 328.622,Z 679.425,A -85,B 0,C 180,E1 -22402.96,E2 -22402.96} C_VEL
LIN {X 0,Y 328.466,Z 687.315,A -85,B 0,C 180,E1 -22405.107,E2 -22405.107} C_VEL
LIN {X 0,Y 328.351,Z 692.712,A -85,B 0,C 180,E1 -22406.943,E2 -22406.943} C_VEL
LIN {X 0,Y 328.3,Z 697.056,A -85,B 0,C 180,E1 -22408.777,E2 -22408.777} C_VEL
LIN {X 0,Y 328.268,Z 699.419,A -85,B 0,C 180,E1 -22410,E2 -22410} C_VEL
LIN {X 0,Y 328.141,Z 702.933,A -85,B 0,C 180,E1 -22412.447,E2 -22412.447} C_VEL
LIN {X 0,Y 328.261,Z 704.986,A -85,B 0,C 180,E1 -22414.896,E2 -22414.896} C_VEL
LIN {X 0,Y 328.858,Z 705.628,A -85,B 0,C 180,E1 -22417.342,E2 -22417.342} C_VEL
LIN {X 0,Y 329.845,Z 704.889,A -85,B 0,C 180,E1 -22419.781,E2 -22419.781} C_VEL
LIN {X 0,Y 331.562,Z 702.776,A -85,B 0,C 180,E1 -22422.196,E2 -22422.196} C_VEL
LIN {X 0,Y 334.053,Z 699.248,A -85,B 0,C 180,E1 -22424.573,E2 -22424.573} C_VEL
LIN {X 0,Y 336.75,Z 694.298,A -85,B 0,C 180,E1 -22426.93,E2 -22426.93} C_VEL
LIN {X 0,Y 340.351,Z 687.725,A -85,B 0,C 180,E1 -22429.225,E2 -22429.225} C_VEL
LIN {X 0,Y 344.052,Z 680.482,A -85,B 0,C 180,E1 -22431.184,E2 -22431.184} C_VEL
LIN {X 0,Y 348.136,Z 671.683,A -85,B 0,C 180,E1 -22433.1,E2 -22433.1} C_VEL
LIN {X 0,Y 352.744,Z 660.965,A -85,B 0,C 180,E1 -22434.958,E2 -22434.958} C_VEL
LIN {X 0,Y 357.474,Z 648.932,A -85,B 0,C 180,E1 -22436.629,E2 -22436.629} C_VEL
LIN {X 0,Y 361.765,Z 636.593,A -85,B 0,C 180,E1 -22438.003,E2 -22438.003} C_VEL
LIN {X 0,Y 366.071,Z 623.018,A -85,B 0,C 180,E1 -22439.204,E2 -22439.204} C_VEL
LIN {X 0,Y 369.723,Z 609.749,A -85,B 0,C 180,E1 -22440.135,E2 -22440.135} C_VEL
LIN {X 0,Y 373.154,Z 595.154,A -85,B 0,C 180,E1 -22440.921,E2 -22440.921} C_VEL
LIN {X 0,Y 376.252,Z 578.163,A -85,B 0,C 180,E1 -22441.612,E2 -22441.612} C_VEL
LIN {X 0,Y 389.569,Z 494.608,A -85,B 0,C 180,E1 -22444.513,E2 -22444.513} C_VEL
LIN {X 0,Y 390.817,Z 480.544,A -85,B 0,C 180,E1 -22445.391,E2 -22445.391} C_VEL
LIN {X 0,Y 391.606,Z 468.8,A -85,B 0,C 180,E1 -22446.271,E2 -22446.271} C_VEL
LIN {X 0,Y 392.32,Z 456.779,A -85,B 0,C 180,E1 -22447.313,E2 -22447.313} C_VEL
LIN {X 0,Y 392.543,Z 451.524,A -85,B 0,C 180,E1 -22447.853,E2 -22447.853} C_VEL
LIN {X 0,Y 389.81,Z 448.58,A -85,B 0,C 180,E1 -22449.868,E2 -22449.868} C_VEL
LIN {X 0,Y 387.864,Z 447.073,A -85,B 0,C 180,E1 -22451.927,E2 -22451.927} C_VEL
LIN {X 0,Y 386.663,Z 447.023,A -85,B 0,C 180,E1 -22454.291,E2 -22454.291} C_VEL
LIN {X 0,Y 386.43,Z 448.353,A -85,B 0,C 180,E1 -22456.032,E2 -22456.032} C_VEL
LIN {X 0,Y 386.945,Z 451.484,A -85,B 0,C 180,E1 -22458.23,E2 -22458.23} C_VEL
LIN {X 0,Y 387.623,Z 454.454,A -85,B 0,C 180,E1 -22459.541,E2 -22459.541} C_VEL
LIN {X 0,Y 388.686,Z 458.685,A -85,B 0,C 180,E1 -22460.991,E2 -22460.991} C_VEL
LIN {X 0,Y 389.521,Z 462.609,A -85,B 0,C 180,E1 -22461.995,E2 -22461.995} C_VEL
LIN {X 0,Y 389.253,Z 478.096,A -85,B 0,C 180,E1 -22463.685,E2 -22463.685} C_VEL
LIN {X 0,Y 389.075,Z 493.181,A -85,B 0,C 180,E1 -22465.1,E2 -22465.1} C_VEL
LIN {X 0,Y 388.846,Z 500.332,A -85,B 0,C 180,E1 -22465.661,E2 -22465.661} C_VEL
LIN {X 0,Y 375.265,Z 585.493,A -85,B 0,C 180,E1 -22468.609,E2 -22468.609} C_VEL
LIN {X 0,Y 372.185,Z 600.23,A -85,B 0,C 180,E1 -22469.304,E2 -22469.304} C_VEL
LIN {X 0,Y 368.431,Z 615.054,A -85,B 0,C 180,E1 -22470.22,E2 -22470.22} C_VEL
LIN {X 0,Y 364.524,Z 628.41,A -85,B 0,C 180,E1 -22471.29,E2 -22471.29} C_VEL
LIN {X 0,Y 360.43,Z 640.733,A -85,B 0,C 180,E1 -22472.513,E2 -22472.513} C_VEL
LIN {X 0,Y 356.632,Z 651.132,A -85,B 0,C 180,E1 -22473.774,E2 -22473.774} C_VEL
LIN {X 0,Y 352.335,Z 661.782,A -85,B 0,C 180,E1 -22475.325,E2 -22475.325} C_VEL
LIN {X 0,Y 347.815,Z 672.086,A -85,B 0,C 180,E1 -22477.191,E2 -22477.191} C_VEL
LIN {X 0,Y 343.742,Z 680.559,A -85,B 0,C 180,E1 -22479.109,E2 -22479.109} C_VEL
LIN {X 0,Y 339.723,Z 688.406,A -85,B 0,C 180,E1 -22481.363,E2 -22481.363} C_VEL
LIN {X 0,Y 336.254,Z 694.56,A -85,B 0,C 180,E1 -22483.667,E2 -22483.667} C_VEL
LIN {X 0,Y 334.295,Z 698.06,A -85,B 0,C 180,E1 -22485.438,E2 -22485.438} C_VEL
LIN {X 0,Y 331.771,Z 701.556,A -85,B 0,C 180,E1 -22487.812,E2 -22487.812} C_VEL
LIN {X 0,Y 329.994,Z 703.644,A -85,B 0,C 180,E1 -22490.224,E2 -22490.224} C_VEL
LIN {X 0,Y 328.923,Z 704.366,A -85,B 0,C 180,E1 -22492.66,E2 -22492.66} C_VEL
LIN {X 0,Y 328.265,Z 703.719,A -85,B 0,C 180,E1 -22495.104,E2 -22495.104} C_VEL
LIN {X 0,Y 328.062,Z 701.67,A -85,B 0,C 180,E1 -22497.553,E2 -22497.553} C_VEL
LIN {X 0,Y 328.166,Z 698.172,A -85,B 0,C 180,E1 -22500,E2 -22500} C_VEL
LIN {X 0,Y 328.208,Z 694.534,A -85,B 0,C 180,E1 -22501.835,E2 -22501.835} C_VEL
LIN {X 0,Y 328.309,Z 689.867,A -85,B 0,C 180,E1 -22503.67,E2 -22503.67} C_VEL
LIN {X 0,Y 328.458,Z 683.085,A -85,B 0,C 180,E1 -22505.814,E2 -22505.814} C_VEL
LIN {X 0,Y 328.704,Z 675.9,A -85,B 0,C 180,E1 -22507.654,E2 -22507.654} C_VEL
LIN {X 0,Y 329.15,Z 667.272,A -85,B 0,C 180,E1 -22509.493,E2 -22509.493} C_VEL
LIN {X 0,Y 329.701,Z 656.82,A -85,B 0,C 180,E1 -22511.334,E2 -22511.334} C_VEL
LIN {X 0,Y 330.494,Z 645.143,A -85,B 0,C 180,E1 -22513.035,E2 -22513.035} C_VEL
LIN {X 0,Y 331.25,Z 632.591,A -85,B 0,C 180,E1 -22514.543,E2 -22514.543} C_VEL
LIN {X 0,Y 332.103,Z 620.242,A -85,B 0,C 180,E1 -22515.757,E2 -22515.757} C_VEL
LIN {X 0,Y 332.954,Z 605.736,A -85,B 0,C 180,E1 -22516.893,E2 -22516.893} C_VEL
LIN {X 0,Y 333.642,Z 590.686,A -85,B 0,C 180,E1 -22517.802,E2 -22517.802} C_VEL
LIN {X 0,Y 334.326,Z 575.07,A -85,B 0,C 180,E1 -22518.475,E2 -22518.475} C_VEL
LIN {X 0,Y 337.614,Z 476.109,A -85,B 0,C 180,E1 -22521.809,E2 -22521.809} C_VEL
LIN {X 0,Y 335.275,Z 447.81,A -85,B 0,C 180,E1 -22522.832,E2 -22522.832} C_VEL
LIN {X 0,Y 335.008,Z 439.387,A -85,B 0,C 180,E1 -22523.164,E2 -22523.164} C_VEL
LIN {X 0,Y 337.345,Z 412.624,A -85,B 0,C 180,E1 -22527.181,E2 -22527.181} C_VEL
LIN {X 0,Y 339.002,Z 395.184,A -85,B 0,C 180,E1 -22529.796,E2 -22529.796} C_VEL
LIN {X 0,Y 338.378,Z 390.951,A -85,B 0,C 180,E1 -22530.474,E2 -22530.474} C_VEL
LIN {X 0,Y 334.228,Z 372.19,A -85,B 0,C 180,E1 -22533.588,E2 -22533.588} C_VEL
LIN {X 0,Y 330.799,Z 356.837,A -85,B 0,C 180,E1 -22536.229,E2 -22536.229} C_VEL
LIN {X 0,Y 330.72,Z 356.844,A -85,B 0,C 180,E1 -22539.449,E2 -22539.449} C_VEL
LIN {X 0,Y 330.737,Z 356.843,A -85,B 0,C 180,E1 -22542.665,E2 -22542.665} C_VEL
LIN {X 0,Y 330.758,Z 356.836,A -85,B 0,C 180,E1 -22546.056,E2 -22546.056} C_VEL
LIN {X 0,Y 330.714,Z 356.84,A -85,B 0,C 180,E1 -22549.683,E2 -22549.683} C_VEL
LIN {X 0,Y 330.745,Z 356.842,A -85,B 0,C 180,E1 -22552.109,E2 -22552.109} C_VEL
LIN {X 0,Y 330.753,Z 356.84,A -85,B 0,C 180,E1 -22555.682,E2 -22555.682} C_VEL
LIN {X 0,Y 330.753,Z 356.836,A -85,B 0,C 180,E1 -22559.452,E2 -22559.452} C_VEL
LIN {X 0,Y 330.791,Z 356.839,A -85,B 0,C 180,E1 -22562.792,E2 -22562.792} C_VEL
LIN {X 0,Y 330.794,Z 356.838,A -85,B 0,C 180,E1 -22566.277,E2 -22566.277} C_VEL
LIN {X 0,Y 330.782,Z 356.839,A -85,B 0,C 180,E1 -22567.554,E2 -22567.554} C_VEL
LIN {X 0,Y 331.919,Z 359.853,A -85,B 0,C 180,E1 -22567.742,E2 -22567.742} C_VEL
LIN {X 0,Y 340.283,Z 377.77,A -85,B 0,C 180,E1 -22568.833,E2 -22568.833} C_VEL
LIN {X 0,Y 346.044,Z 391.675,A -85,B 0,C 180,E1 -22569.583,E2 -22569.583} C_VEL
LIN {X 0,Y 344.412,Z 462.941,A -85,B 0,C 180,E1 -22571.049,E2 -22571.049} C_VEL
LIN {X 0,Y 344.217,Z 478.712,A -85,B 0,C 180,E1 -22571.461,E2 -22571.461} C_VEL
LIN {X 0,Y 343.649,Z 492.69,A -85,B 0,C 180,E1 -22572.044,E2 -22572.044} C_VEL
LIN {X 0,Y 342.75,Z 506.223,A -85,B 0,C 180,E1 -22572.84,E2 -22572.84} C_VEL
LIN {X 0,Y 341.655,Z 518.418,A -85,B 0,C 180,E1 -22573.78,E2 -22573.78} C_VEL
LIN {X 0,Y 340.448,Z 530.396,A -85,B 0,C 180,E1 -22574.945,E2 -22574.945} C_VEL
LIN {X 0,Y 338.972,Z 542.381,A -85,B 0,C 180,E1 -22576.386,E2 -22576.386} C_VEL
LIN {X 0,Y 337.245,Z 553.4,A -85,B 0,C 180,E1 -22578.013,E2 -22578.013} C_VEL
LIN {X 0,Y 335.637,Z 563.18,A -85,B 0,C 180,E1 -22579.783,E2 -22579.783} C_VEL
LIN {X 0,Y 334.24,Z 571.305,A -85,B 0,C 180,E1 -22581.565,E2 -22581.565} C_VEL
LIN {X 0,Y 333.085,Z 578.087,A -85,B 0,C 180,E1 -22583.359,E2 -22583.359} C_VEL
LIN {X 0,Y 332.047,Z 583.724,A -85,B 0,C 180,E1 -22585.16,E2 -22585.16} C_VEL
LIN {X 0,Y 331.291,Z 588.325,A -85,B 0,C 180,E1 -22586.97,E2 -22586.97} C_VEL
LIN {X 0,Y 330.573,Z 593.107,A -85,B 0,C 180,E1 -22589.393,E2 -22589.393} C_VEL
LIN {X 0,Y 330.253,Z 595.724,A -85,B 0,C 180,E1 -22591.215,E2 -22591.215} C_VEL
LIN {X 0,Y 330.072,Z 598.033,A -85,B 0,C 180,E1 -22593.65,E2 -22593.65} C_VEL
LIN {X 0,Y 330.23,Z 599.036,A -85,B 0,C 180,E1 -22596.088,E2 -22596.088} C_VEL
LIN {X 0,Y 330.588,Z 598.76,A -85,B 0,C 180,E1 -22598.53,E2 -22598.53} C_VEL
LIN {X 0,Y 331.206,Z 597.19,A -85,B 0,C 180,E1 -22600.973,E2 -22600.973} C_VEL
LIN {X 0,Y 332.37,Z 594.253,A -85,B 0,C 180,E1 -22603.404,E2 -22603.404} C_VEL
LIN {X 0,Y 333.829,Z 589.883,A -85,B 0,C 180,E1 -22605.829,E2 -22605.829} C_VEL
LIN {X 0,Y 335.182,Z 585.519,A -85,B 0,C 180,E1 -22607.639,E2 -22607.639} C_VEL
LIN {X 0,Y 336.721,Z 580.192,A -85,B 0,C 180,E1 -22609.441,E2 -22609.441} C_VEL
LIN {X 0,Y 338.831,Z 572.546,A -85,B 0,C 180,E1 -22611.524,E2 -22611.524} C_VEL
LIN {X 0,Y 340.91,Z 564.5,A -85,B 0,C 180,E1 -22613.298,E2 -22613.298} C_VEL
LIN {X 0,Y 343.203,Z 554.783,A -85,B 0,C 180,E1 -22615.055,E2 -22615.055} C_VEL
LIN {X 0,Y 345.433,Z 543.75,A -85,B 0,C 180,E1 -22616.687,E2 -22616.687} C_VEL
LIN {X 0,Y 347.615,Z 531.862,A -85,B 0,C 180,E1 -22618.1,E2 -22618.1} C_VEL
LIN {X 0,Y 349.467,Z 519.831,A -85,B 0,C 180,E1 -22619.246,E2 -22619.246} C_VEL
LIN {X 0,Y 350.831,Z 506.907,A -85,B 0,C 180,E1 -22620.238,E2 -22620.238} C_VEL
LIN {X 0,Y 352.004,Z 492.772,A -85,B 0,C 180,E1 -22621.049,E2 -22621.049} C_VEL
LIN {X 0,Y 352.735,Z 477.987,A -85,B 0,C 180,E1 -22621.643,E2 -22621.643} C_VEL
LIN {X 0,Y 353.158,Z 458.837,A -85,B 0,C 180,E1 -22622.102,E2 -22622.102} C_VEL
LIN {X 0,Y 354.953,Z 403.049,A -85,B 0,C 180,E1 -22623.218,E2 -22623.218} C_VEL
LIN {X 0,Y 347.183,Z 387.01,A -85,B 0,C 180,E1 -22624.379,E2 -22624.379} C_VEL
LIN {X 0,Y 336.619,Z 367.689,A -85,B 0,C 180,E1 -22626.009,E2 -22626.009} C_VEL
LIN {X 0,Y 332.094,Z 360.262,A -85,B 0,C 180,E1 -22626.727,E2 -22626.727} C_VEL
LIN {X 0,Y 330.857,Z 357.582,A -85,B 0,C 180,E1 -22626.945,E2 -22626.945} C_VEL
LIN {X 0,Y 330.721,Z 356.848,A -85,B 0,C 180,E1 -22627.014,E2 -22627.014} C_VEL
LIN {X 0,Y 330.7,Z 356.853,A -85,B 0,C 180,E1 -22631.042,E2 -22631.042} C_VEL
LIN {X 0,Y 330.69,Z 356.848,A -85,B 0,C 180,E1 -22634.346,E2 -22634.346} C_VEL
LIN {X 0,Y 330.705,Z 356.843,A -85,B 0,C 180,E1 -22637.844,E2 -22637.844} C_VEL
LIN {X 0,Y 330.702,Z 356.82,A -85,B 0,C 180,E1 -22641.599,E2 -22641.599} C_VEL
LIN {X 0,Y 330.728,Z 356.818,A -85,B 0,C 180,E1 -22645.122,E2 -22645.122} C_VEL
LIN {X 0,Y 330.723,Z 356.84,A -85,B 0,C 180,E1 -22648.029,E2 -22648.029} C_VEL
LIN {X 0,Y 330.737,Z 356.84,A -85,B 0,C 180,E1 -22650.849,E2 -22650.849} C_VEL
LIN {X 0,Y 330.76,Z 356.837,A -85,B 0,C 180,E1 -22652.459,E2 -22652.459} C_VEL
LIN {X 0,Y 330.099,Z 356.918,A -85,B 0,C 180,E1 -22653.136,E2 -22653.136} C_VEL
LIN {X 0,Y 327.254,Z 357.272,A -85,B 0,C 180,E1 -22654.198,E2 -22654.198} C_VEL
LIN {X 0,Y 324.389,Z 357.63,A -85,B 0,C 180,E1 -22655.277,E2 -22655.277} C_VEL
LIN {X 0,Y 323.726,Z 357.715,A -85,B 0,C 180,E1 -22655.975,E2 -22655.975} C_VEL
LIN {X 0,Y 323.751,Z 357.715,A -85,B 0,C 180,E1 -22656.975,E2 -22656.975} C_VEL
LIN {X 0,Y 329.893,Z 381.782,A -85,B 0,C 180,E1 -22657.955,E2 -22657.955} C_VEL
LIN {X 0,Y 327.263,Z 474.44,A -85,B 0,C 180,E1 -22661.113,E2 -22661.113} C_VEL
LIN {X 0,Y 326.858,Z 488.755,A -85,B 0,C 180,E1 -22661.816,E2 -22661.816} C_VEL
LIN {X 0,Y 326.329,Z 503.167,A -85,B 0,C 180,E1 -22662.754,E2 -22662.754} C_VEL
LIN {X 0,Y 325.6,Z 517.167,A -85,B 0,C 180,E1 -22663.92,E2 -22663.92} C_VEL
LIN {X 0,Y 324.856,Z 530.694,A -85,B 0,C 180,E1 -22665.324,E2 -22665.324} C_VEL
LIN {X 0,Y 324.185,Z 543.687,A -85,B 0,C 180,E1 -22666.965,E2 -22666.965} C_VEL
LIN {X 0,Y 323.553,Z 555.357,A -85,B 0,C 180,E1 -22668.764,E2 -22668.764} C_VEL
LIN {X 0,Y 322.956,Z 565.491,A -85,B 0,C 180,E1 -22670.638,E2 -22670.638} C_VEL
LIN {X 0,Y 322.615,Z 573.972,A -85,B 0,C 180,E1 -22672.515,E2 -22672.515} C_VEL
LIN {X 0,Y 322.427,Z 582.194,A -85,B 0,C 180,E1 -22674.702,E2 -22674.702} C_VEL
LIN {X 0,Y 322.493,Z 588.82,A -85,B 0,C 180,E1 -22676.887,E2 -22676.887} C_VEL
LIN {X 0,Y 322.724,Z 594.704,A -85,B 0,C 180,E1 -22679.378,E2 -22679.378} C_VEL
LIN {X 0,Y 323.191,Z 598.109,A -85,B 0,C 180,E1 -22681.242,E2 -22681.242} C_VEL
LIN {X 0,Y 324.164,Z 601.312,A -85,B 0,C 180,E1 -22683.716,E2 -22683.716} C_VEL
LIN {X 0,Y 325.599,Z 603.114,A -85,B 0,C 180,E1 -22686.175,E2 -22686.175} C_VEL
LIN {X 0,Y 327.371,Z 603.544,A -85,B 0,C 180,E1 -22688.613,E2 -22688.613} C_VEL
LIN {X 0,Y 329.773,Z 602.568,A -85,B 0,C 180,E1 -22691.02,E2 -22691.02} C_VEL
LIN {X 0,Y 332.971,Z 600.077,A -85,B 0,C 180,E1 -22693.379,E2 -22693.379} C_VEL
LIN {X 0,Y 336.406,Z 596.163,A -85,B 0,C 180,E1 -22695.704,E2 -22695.704} C_VEL
LIN {X 0,Y 340.281,Z 590.695,A -85,B 0,C 180,E1 -22697.985,E2 -22697.985} C_VEL
LIN {X 0,Y 343.494,Z 585.44,A -85,B 0,C 180,E1 -22699.661,E2 -22699.661} C_VEL
LIN {X 0,Y 347.815,Z 577.397,A -85,B 0,C 180,E1 -22701.718,E2 -22701.718} C_VEL
LIN {X 0,Y 351.866,Z 568.761,A -85,B 0,C 180,E1 -22703.461,E2 -22703.461} C_VEL
LIN {X 0,Y 355.949,Z 559.167,A -85,B 0,C 180,E1 -22705.029,E2 -22705.029} C_VEL
LIN {X 0,Y 360.184,Z 547.602,A -85,B 0,C 180,E1 -22706.569,E2 -22706.569} C_VEL
LIN {X 0,Y 364.302,Z 534.678,A -85,B 0,C 180,E1 -22707.947,E2 -22707.947} C_VEL
LIN {X 0,Y 367.618,Z 521.928,A -85,B 0,C 180,E1 -22709.069,E2 -22709.069} C_VEL
LIN {X 0,Y 370.252,Z 509.744,A -85,B 0,C 180,E1 -22709.931,E2 -22709.931} C_VEL
LIN {X 0,Y 372.764,Z 495.126,A -85,B 0,C 180,E1 -22710.761,E2 -22710.761} C_VEL
LIN {X 0,Y 376.363,Z 469.074,A -85,B 0,C 180,E1 -22711.818,E2 -22711.818} C_VEL
LIN {X 0,Y 382.161,Z 432.638,A -85,B 0,C 180,E1 -22713.09,E2 -22713.09} C_VEL
LIN {X 0,Y 379.403,Z 426.768,A -85,B 0,C 180,E1 -22714.687,E2 -22714.687} C_VEL
LIN {X 0,Y 377.479,Z 423.151,A -85,B 0,C 180,E1 -22715.964,E2 -22715.964} C_VEL
LIN {X 0,Y 375.845,Z 420.024,A -85,B 0,C 180,E1 -22717.271,E2 -22717.271} C_VEL
LIN {X 0,Y 374.078,Z 416.54,A -85,B 0,C 180,E1 -22719.203,E2 -22719.203} C_VEL
LIN {X 0,Y 372.465,Z 414.923,A -85,B 0,C 180,E1 -22721.856,E2 -22721.856} C_VEL
LIN {X 0,Y 372.292,Z 414.748,A -85,B 0,C 180,E1 -22724.361,E2 -22724.361} C_VEL
LIN {X 0,Y 373.601,Z 416.315,A -85,B 0,C 180,E1 -22727.231,E2 -22727.231} C_VEL
LIN {X 0,Y 375.595,Z 420.346,A -85,B 0,C 180,E1 -22729.535,E2 -22729.535} C_VEL
LIN {X 0,Y 375.939,Z 425.051,A -85,B 0,C 180,E1 -22730.451,E2 -22730.451} C_VEL
LIN {X 0,Y 376.797,Z 435.127,A -85,B 0,C 180,E1 -22732.108,E2 -22732.108} C_VEL
LIN {X 0,Y 376.017,Z 453.197,A -85,B 0,C 180,E1 -22733.656,E2 -22733.656} C_VEL
LIN {X 0,Y 375.274,Z 470.579,A -85,B 0,C 180,E1 -22734.965,E2 -22734.965} C_VEL
LIN {X 0,Y 374.523,Z 483.17,A -85,B 0,C 180,E1 -22735.788,E2 -22735.788} C_VEL
LIN {X 0,Y 373.5,Z 494.726,A -85,B 0,C 180,E1 -22736.386,E2 -22736.386} C_VEL
LIN {X 0,Y 367.589,Z 533.571,A -85,B 0,C 180,E1 -22737.754,E2 -22737.754} C_VEL
LIN {X 0,Y 363.889,Z 550.974,A -85,B 0,C 180,E1 -22738.525,E2 -22738.525} C_VEL
LIN {X 0,Y 359.686,Z 566.408,A -85,B 0,C 180,E1 -22739.419,E2 -22739.419} C_VEL
LIN {X 0,Y 355.253,Z 580.416,A -85,B 0,C 180,E1 -22740.467,E2 -22740.467} C_VEL
LIN {X 0,Y 350.845,Z 592.874,A -85,B 0,C 180,E1 -22741.619,E2 -22741.619} C_VEL
LIN {X 0,Y 346.345,Z 604.395,A -85,B 0,C 180,E1 -22742.932,E2 -22742.932} C_VEL
LIN {X 0,Y 341.192,Z 616.673,A -85,B 0,C 180,E1 -22744.685,E2 -22744.685} C_VEL
LIN {X 0,Y 336.958,Z 626.454,A -85,B 0,C 180,E1 -22746.412,E2 -22746.412} C_VEL
LIN {X 0,Y 333.419,Z 634.307,A -85,B 0,C 180,E1 -22748.106,E2 -22748.106} C_VEL
LIN {X 0,Y 329.816,Z 642.096,A -85,B 0,C 180,E1 -22750.135,E2 -22750.135} C_VEL
LIN {X 0,Y 327.289,Z 647.659,A -85,B 0,C 180,E1 -22751.921,E2 -22751.921} C_VEL
LIN {X 0,Y 324.753,Z 653.685,A -85,B 0,C 180,E1 -22754.359,E2 -22754.359} C_VEL
LIN {X 0,Y 323.45,Z 657.276,A -85,B 0,C 180,E1 -22756.219,E2 -22756.219} C_VEL
LIN {X 0,Y 322.369,Z 660.819,A -85,B 0,C 180,E1 -22758.723,E2 -22758.723} C_VEL
LIN {X 0,Y 322.272,Z 661.875,A -85,B 0,C 180,E1 -22759.551,E2 -22759.551} C_VEL
LIN {X 0,Y 321.871,Z 670.772,A -85,B 0,C 180,E1 -22761.238,E2 -22761.238} C_VEL
LIN {X 0,Y 321.579,Z 679.091,A -85,B 0,C 180,E1 -22763.119,E2 -22763.119} C_VEL
LIN {X 0,Y 321.426,Z 687.035,A -85,B 0,C 180,E1 -22765.312,E2 -22765.312} C_VEL
LIN {X 0,Y 321.259,Z 693.291,A -85,B 0,C 180,E1 -22767.501,E2 -22767.501} C_VEL
LIN {X 0,Y 321.221,Z 697.48,A -85,B 0,C 180,E1 -22769.375,E2 -22769.375} C_VEL
LIN {X 0,Y 321.083,Z 700.728,A -85,B 0,C 180,E1 -22771.25,E2 -22771.25} C_VEL
LIN {X 0,Y 321.077,Z 703.718,A -85,B 0,C 180,E1 -22773.752,E2 -22773.752} C_VEL
LIN {X 0,Y 321.437,Z 705.296,A -85,B 0,C 180,E1 -22776.255,E2 -22776.255} C_VEL
LIN {X 0,Y 322.233,Z 705.498,A -85,B 0,C 180,E1 -22778.752,E2 -22778.752} C_VEL
LIN {X 0,Y 323.667,Z 704.346,A -85,B 0,C 180,E1 -22781.231,E2 -22781.231} C_VEL
LIN {X 0,Y 325.903,Z 701.823,A -85,B 0,C 180,E1 -22783.675,E2 -22783.675} C_VEL
LIN {X 0,Y 328.634,Z 697.898,A -85,B 0,C 180,E1 -22786.086,E2 -22786.086} C_VEL
LIN {X 0,Y 330.932,Z 693.977,A -85,B 0,C 180,E1 -22787.873,E2 -22787.873} C_VEL
LIN {X 0,Y 334.831,Z 687.357,A -85,B 0,C 180,E1 -22790.192,E2 -22790.192} C_VEL
LIN {X 0,Y 338.793,Z 680.068,A -85,B 0,C 180,E1 -22792.167,E2 -22792.167} C_VEL
LIN {X 0,Y 343.196,Z 671.205,A -85,B 0,C 180,E1 -22794.091,E2 -22794.091} C_VEL
LIN {X 0,Y 348.095,Z 660.464,A -85,B 0,C 180,E1 -22795.954,E2 -22795.954} C_VEL
LIN {X 0,Y 353.109,Z 648.387,A -85,B 0,C 180,E1 -22797.625,E2 -22797.625} C_VEL
LIN {X 0,Y 357.64,Z 636.035,A -85,B 0,C 180,E1 -22798.995,E2 -22798.995} C_VEL
LIN {X 0,Y 362.163,Z 622.464,A -85,B 0,C 180,E1 -22800.189,E2 -22800.189} C_VEL
LIN {X 0,Y 366,Z 609.158,A -85,B 0,C 180,E1 -22801.113,E2 -22801.113} C_VEL
LIN {X 0,Y 369.556,Z 594.606,A -85,B 0,C 180,E1 -22801.893,E2 -22801.893} C_VEL
LIN {X 0,Y 372.789,Z 577.689,A -85,B 0,C 180,E1 -22802.577,E2 -22802.577} C_VEL
LIN {X 0,Y 386.436,Z 496.54,A -85,B 0,C 180,E1 -22805.412,E2 -22805.412} C_VEL
LIN {X 0,Y 387.799,Z 483.558,A -85,B 0,C 180,E1 -22806.226,E2 -22806.226} C_VEL
LIN {X 0,Y 388.815,Z 471.531,A -85,B 0,C 180,E1 -22807.142,E2 -22807.142} C_VEL
LIN {X 0,Y 389.704,Z 460.227,A -85,B 0,C 180,E1 -22808.142,E2 -22808.142} C_VEL
LIN {X 0,Y 389.895,Z 457.495,A -85,B 0,C 180,E1 -22808.424,E2 -22808.424} C_VEL
LIN {X 0,Y 387.489,Z 454.961,A -85,B 0,C 180,E1 -22810.385,E2 -22810.385} C_VEL
LIN {X 0,Y 385.934,Z 453.845,A -85,B 0,C 180,E1 -22812.185,E2 -22812.185} C_VEL
LIN {X 0,Y 384.932,Z 453.91,A -85,B 0,C 180,E1 -22814.283,E2 -22814.283} C_VEL
LIN {X 0,Y 384.681,Z 455.517,A -85,B 0,C 180,E1 -22816.218,E2 -22816.218} C_VEL
LIN {X 0,Y 385.274,Z 459.09,A -85,B 0,C 180,E1 -22818.496,E2 -22818.496} C_VEL
LIN {X 0,Y 386.375,Z 464.419,A -85,B 0,C 180,E1 -22820.475,E2 -22820.475} C_VEL
LIN {X 0,Y 386.961,Z 467.862,A -85,B 0,C 180,E1 -22821.363,E2 -22821.363} C_VEL
LIN {X 0,Y 386.368,Z 482.19,A -85,B 0,C 180,E1 -22822.933,E2 -22822.933} C_VEL
LIN {X 0,Y 385.916,Z 496.541,A -85,B 0,C 180,E1 -22824.299,E2 -22824.299} C_VEL
LIN {X 0,Y 385.599,Z 502.347,A -85,B 0,C 180,E1 -22824.756,E2 -22824.756} C_VEL
LIN {X 0,Y 371.643,Z 585.559,A -85,B 0,C 180,E1 -22827.671,E2 -22827.671} C_VEL
LIN {X 0,Y 368.542,Z 599.666,A -85,B 0,C 180,E1 -22828.33,E2 -22828.33} C_VEL
LIN {X 0,Y 364.582,Z 614.524,A -85,B 0,C 180,E1 -22829.235,E2 -22829.235} C_VEL
LIN {X 0,Y 360.493,Z 627.906,A -85,B 0,C 180,E1 -22830.299,E2 -22830.299} C_VEL
LIN {X 0,Y 356.201,Z 640.223,A -85,B 0,C 180,E1 -22831.52,E2 -22831.52} C_VEL
LIN {X 0,Y 352.16,Z 650.658,A -85,B 0,C 180,E1 -22832.776,E2 -22832.776} C_VEL
LIN {X 0,Y 347.621,Z 661.324,A -85,B 0,C 180,E1 -22834.328,E2 -22834.328} C_VEL
LIN {X 0,Y 342.809,Z 671.69,A -85,B 0,C 180,E1 -22836.2,E2 -22836.2} C_VEL
LIN {X 0,Y 338.453,Z 680.201,A -85,B 0,C 180,E1 -22838.129,E2 -22838.129} C_VEL
LIN {X 0,Y 335.201,Z 686.303,A -85,B 0,C 180,E1 -22839.831,E2 -22839.831} C_VEL
LIN {X 0,Y 331.253,Z 692.875,A -85,B 0,C 180,E1 -22842.145,E2 -22842.145} C_VEL
LIN {X 0,Y 328.898,Z 696.766,A -85,B 0,C 180,E1 -22843.928,E2 -22843.928} C_VEL
LIN {X 0,Y 326.072,Z 700.671,A -85,B 0,C 180,E1 -22846.332,E2 -22846.332} C_VEL
LIN {X 0,Y 323.867,Z 703.16,A -85,B 0,C 180,E1 -22848.776,E2 -22848.776} C_VEL
LIN {X 0,Y 322.36,Z 704.291,A -85,B 0,C 180,E1 -22851.252,E2 -22851.252} C_VEL
LIN {X 0,Y 321.471,Z 704.074,A -85,B 0,C 180,E1 -22853.746,E2 -22853.746} C_VEL
LIN {X 0,Y 321.067,Z 702.492,A -85,B 0,C 180,E1 -22856.248,E2 -22856.248} C_VEL
LIN {X 0,Y 321.023,Z 699.512,A -85,B 0,C 180,E1 -22858.75,E2 -22858.75} C_VEL
LIN {X 0,Y 321.124,Z 696.287,A -85,B 0,C 180,E1 -22860.625,E2 -22860.625} C_VEL
LIN {X 0,Y 321.201,Z 692.135,A -85,B 0,C 180,E1 -22862.5,E2 -22862.5} C_VEL
LIN {X 0,Y 321.337,Z 686.915,A -85,B 0,C 180,E1 -22864.376,E2 -22864.376} C_VEL
LIN {X 0,Y 321.518,Z 679.377,A -85,B 0,C 180,E1 -22866.568,E2 -22866.568} C_VEL
LIN {X 0,Y 321.799,Z 671.447,A -85,B 0,C 180,E1 -22868.449,E2 -22868.449} C_VEL
LIN {X 0,Y 322.361,Z 661.932,A -85,B 0,C 180,E1 -22870.327,E2 -22870.327} C_VEL
LIN {X 0,Y 323.048,Z 650.368,A -85,B 0,C 180,E1 -22872.205,E2 -22872.205} C_VEL
LIN {X 0,Y 323.803,Z 638.735,A -85,B 0,C 180,E1 -22873.766,E2 -22873.766} C_VEL
LIN {X 0,Y 324.61,Z 626.096,A -85,B 0,C 180,E1 -22875.167,E2 -22875.167} C_VEL
LIN {X 0,Y 325.508,Z 612.206,A -85,B 0,C 180,E1 -22876.406,E2 -22876.406} C_VEL
LIN {X 0,Y 326.236,Z 596.625,A -85,B 0,C 180,E1 -22877.493,E2 -22877.493} C_VEL
LIN {X 0,Y 326.987,Z 581.694,A -85,B 0,C 180,E1 -22878.258,E2 -22878.258} C_VEL
LIN {X 0,Y 330.577,Z 476.353,A -85,B 0,C 180,E1 -22881.949,E2 -22881.949} C_VEL
LIN {X 0,Y 328.263,Z 448.541,A -85,B 0,C 180,E1 -22882.977,E2 -22882.977} C_VEL
LIN {X 0,Y 327.993,Z 439.534,A -85,B 0,C 180,E1 -22883.323,E2 -22883.323} C_VEL
LIN {X 0,Y 330.298,Z 413.627,A -85,B 0,C 180,E1 -22887.275,E2 -22887.275} C_VEL
LIN {X 0,Y 331.968,Z 395.057,A -85,B 0,C 180,E1 -22890.107,E2 -22890.107} C_VEL
LIN {X 0,Y 328.065,Z 376.851,A -85,B 0,C 180,E1 -22893.159,E2 -22893.159} C_VEL
LIN {X 0,Y 323.76,Z 357.715,A -85,B 0,C 180,E1 -22896.478,E2 -22896.478} C_VEL
LIN {X 0,Y 323.668,Z 357.72,A -85,B 0,C 180,E1 -22900.484,E2 -22900.484} C_VEL
LIN {X 0,Y 323.719,Z 357.717,A -85,B 0,C 180,E1 -22903.821,E2 -22903.821} C_VEL
LIN {X 0,Y 323.703,Z 357.721,A -85,B 0,C 180,E1 -22907.368,E2 -22907.368} C_VEL
LIN {X 0,Y 323.704,Z 357.721,A -85,B 0,C 180,E1 -22911.168,E2 -22911.168} C_VEL
LIN {X 0,Y 323.728,Z 357.716,A -85,B 0,C 180,E1 -22915.306,E2 -22915.306} C_VEL
LIN {X 0,Y 323.689,Z 357.707,A -85,B 0,C 180,E1 -22918.712,E2 -22918.712} C_VEL
LIN {X 0,Y 323.737,Z 357.716,A -85,B 0,C 180,E1 -22922.51,E2 -22922.51} C_VEL
LIN {X 0,Y 323.769,Z 357.714,A -85,B 0,C 180,E1 -22926.408,E2 -22926.408} C_VEL
LIN {X 0,Y 323.751,Z 357.715,A -85,B 0,C 180,E1 -22926.975,E2 -22926.975} C_VEL
LIN {X 0,Y 324.829,Z 360.698,A -85,B 0,C 180,E1 -22927.154,E2 -22927.154} C_VEL
LIN {X 0,Y 333.586,Z 379.045,A -85,B 0,C 180,E1 -22928.33,E2 -22928.33} C_VEL
LIN {X 0,Y 339.448,Z 393.167,A -85,B 0,C 180,E1 -22929.119,E2 -22929.119} C_VEL
LIN {X 0,Y 337.852,Z 464.785,A -85,B 0,C 180,E1 -22930.627,E2 -22930.627} C_VEL
LIN {X 0,Y 337.578,Z 480.189,A -85,B 0,C 180,E1 -22931.043,E2 -22931.043} C_VEL
LIN {X 0,Y 337.032,Z 494.656,A -85,B 0,C 180,E1 -22931.679,E2 -22931.679} C_VEL
LIN {X 0,Y 335.999,Z 508.875,A -85,B 0,C 180,E1 -22932.562,E2 -22932.562} C_VEL
LIN {X 0,Y 334.765,Z 521.48,A -85,B 0,C 180,E1 -22933.593,E2 -22933.593} C_VEL
LIN {X 0,Y 333.397,Z 534.276,A -85,B 0,C 180,E1 -22934.931,E2 -22934.931} C_VEL
LIN {X 0,Y 331.936,Z 545.239,A -85,B 0,C 180,E1 -22936.339,E2 -22936.339} C_VEL
LIN {X 0,Y 330.106,Z 556.266,A -85,B 0,C 180,E1 -22938.06,E2 -22938.06} C_VEL
LIN {X 0,Y 328.458,Z 565.701,A -85,B 0,C 180,E1 -22939.867,E2 -22939.867} C_VEL
LIN {X 0,Y 327.126,Z 573.515,A -85,B 0,C 180,E1 -22941.69,E2 -22941.69} C_VEL
LIN {X 0,Y 325.685,Z 581.039,A -85,B 0,C 180,E1 -22943.827,E2 -22943.827} C_VEL
LIN {X 0,Y 324.774,Z 586.27,A -85,B 0,C 180,E1 -22945.671,E2 -22945.671} C_VEL
LIN {X 0,Y 323.831,Z 591.797,A -85,B 0,C 180,E1 -22948.141,E2 -22948.141} C_VEL
LIN {X 0,Y 323.444,Z 594.917,A -85,B 0,C 180,E1 -22950,E2 -22950} C_VEL
LIN {X 0,Y 323.037,Z 597.871,A -85,B 0,C 180,E1 -22952.486,E2 -22952.486} C_VEL
LIN {X 0,Y 323.072,Z 599.488,A -85,B 0,C 180,E1 -22954.975,E2 -22954.975} C_VEL
LIN {X 0,Y 323.338,Z 599.822,A -85,B 0,C 180,E1 -22957.469,E2 -22957.469} C_VEL
LIN {X 0,Y 323.876,Z 598.869,A -85,B 0,C 180,E1 -22959.963,E2 -22959.963} C_VEL
LIN {X 0,Y 324.783,Z 596.595,A -85,B 0,C 180,E1 -22962.455,E2 -22962.455} C_VEL
LIN {X 0,Y 326.2,Z 592.919,A -85,B 0,C 180,E1 -22964.932,E2 -22964.932} C_VEL
LIN {X 0,Y 327.923,Z 587.705,A -85,B 0,C 180,E1 -22967.4,E2 -22967.4} C_VEL
LIN {X 0,Y 329.469,Z 582.687,A -85,B 0,C 180,E1 -22969.24,E2 -22969.24} C_VEL
LIN {X 0,Y 331.293,Z 576.567,A -85,B 0,C 180,E1 -22971.065,E2 -22971.065} C_VEL
LIN {X 0,Y 333.258,Z 569.206,A -85,B 0,C 180,E1 -22972.882,E2 -22972.882} C_VEL
LIN {X 0,Y 335.515,Z 560.327,A -85,B 0,C 180,E1 -22974.679,E2 -22974.679} C_VEL
LIN {X 0,Y 338.019,Z 549.53,A -85,B 0,C 180,E1 -22976.457,E2 -22976.457} C_VEL
LIN {X 0,Y 340.146,Z 538.568,A -85,B 0,C 180,E1 -22977.93,E2 -22977.93} C_VEL
LIN {X 0,Y 342.303,Z 526.328,A -85,B 0,C 180,E1 -22979.246,E2 -22979.246} C_VEL
LIN {X 0,Y 343.915,Z 514.549,A -85,B 0,C 180,E1 -22980.27,E2 -22980.27} C_VEL
LIN {X 0,Y 345.132,Z 502.33,A -85,B 0,C 180,E1 -22981.121,E2 -22981.121} C_VEL
LIN {X 0,Y 346.134,Z 488.332,A -85,B 0,C 180,E1 -22981.845,E2 -22981.845} C_VEL
LIN {X 0,Y 346.711,Z 473.987,A -85,B 0,C 180,E1 -22982.345,E2 -22982.345} C_VEL
LIN {X 0,Y 348.435,Z 417.803,A -85,B 0,C 180,E1 -22983.518,E2 -22983.518} C_VEL
LIN {X 0,Y 348.724,Z 404.937,A -85,B 0,C 180,E1 -22983.793,E2 -22983.793} C_VEL
LIN {X 0,Y 340.707,Z 388.494,A -85,B 0,C 180,E1 -22985.034,E2 -22985.034} C_VEL
LIN {X 0,Y 331.277,Z 371.405,A -85,B 0,C 180,E1 -22986.537,E2 -22986.537} C_VEL
LIN {X 0,Y 325.325,Z 361.454,A -85,B 0,C 180,E1 -22987.524,E2 -22987.524} C_VEL
LIN {X 0,Y 323.906,Z 358.887,A -85,B 0,C 180,E1 -22987.772,E2 -22987.772} C_VEL
LIN {X 0,Y 323.66,Z 357.725,A -85,B 0,C 180,E1 -22987.86,E2 -22987.86} C_VEL
LIN {X 0,Y 323.668,Z 357.73,A -85,B 0,C 180,E1 -22990.761,E2 -22990.761} C_VEL
LIN {X 0,Y 323.648,Z 357.725,A -85,B 0,C 180,E1 -22994.422,E2 -22994.422} C_VEL
LIN {X 0,Y 323.659,Z 357.72,A -85,B 0,C 180,E1 -22997.864,E2 -22997.864} C_VEL
LIN {X 0,Y 323.641,Z 357.708,A -85,B 0,C 180,E1 -23001.182,E2 -23001.182} C_VEL
LIN {X 0,Y 323.679,Z 357.68,A -85,B 0,C 180,E1 -23004.247,E2 -23004.247} C_VEL
LIN {X 0,Y 323.69,Z 357.721,A -85,B 0,C 180,E1 -23007.559,E2 -23007.559} C_VEL
LIN {X 0,Y 323.678,Z 357.723,A -85,B 0,C 180,E1 -23011.57,E2 -23011.57} C_VEL
LIN {X 0,Y 323.709,Z 357.706,A -85,B 0,C 180,E1 -23014.357,E2 -23014.357} C_VEL
LIN {X 0,Y 323.726,Z 357.715,A -85,B 0,C 180,E1 -23015.975,E2 -23015.975} C_VEL
LIN {X 0,Y 323.73,Z 358.576,A -85,B 0,C 180,E1 -23016.425,E2 -23016.425} C_VEL
LIN {X 0,Y 323.717,Z 360.524,A -85,B 0,C 180,E1 -23016.783,E2 -23016.783} C_VEL
LIN {X 0,Y 323.677,Z 363.562,A -85,B 0,C 180,E1 -23017.082,E2 -23017.082} C_VEL
LIN {X 0,Y 323.57,Z 368.682,A -85,B 0,C 180,E1 -23017.349,E2 -23017.349} C_VEL
LIN {X 0,Y 322.664,Z 387.019,A -85,B 0,C 180,E1 -23017.988,E2 -23017.988} C_VEL
LIN {X 0,Y 320.19,Z 474.318,A -85,B 0,C 180,E1 -23021.051,E2 -23021.051} C_VEL
LIN {X 0,Y 319.742,Z 489.451,A -85,B 0,C 180,E1 -23021.81,E2 -23021.81} C_VEL
LIN {X 0,Y 319.138,Z 504.875,A -85,B 0,C 180,E1 -23022.846,E2 -23022.846} C_VEL
LIN {X 0,Y 318.432,Z 518.663,A -85,B 0,C 180,E1 -23024.04,E2 -23024.04} C_VEL
LIN {X 0,Y 317.697,Z 532.099,A -85,B 0,C 180,E1 -23025.475,E2 -23025.475} C_VEL
LIN {X 0,Y 317.095,Z 543.794,A -85,B 0,C 180,E1 -23026.988,E2 -23026.988} C_VEL
LIN {X 0,Y 316.436,Z 555.615,A -85,B 0,C 180,E1 -23028.832,E2 -23028.832} C_VEL
LIN {X 0,Y 315.861,Z 565.827,A -85,B 0,C 180,E1 -23030.748,E2 -23030.748} C_VEL
LIN {X 0,Y 315.496,Z 574.413,A -85,B 0,C 180,E1 -23032.665,E2 -23032.665} C_VEL
LIN {X 0,Y 315.348,Z 582.707,A -85,B 0,C 180,E1 -23034.902,E2 -23034.902} C_VEL
LIN {X 0,Y 315.393,Z 588.532,A -85,B 0,C 180,E1 -23036.817,E2 -23036.817} C_VEL
LIN {X 0,Y 315.539,Z 593.352,A -85,B 0,C 180,E1 -23038.728,E2 -23038.728} C_VEL
LIN {X 0,Y 316.123,Z 598.355,A -85,B 0,C 180,E1 -23041.269,E2 -23041.269} C_VEL
LIN {X 0,Y 317.102,Z 601.869,A -85,B 0,C 180,E1 -23043.799,E2 -23043.799} C_VEL
LIN {X 0,Y 318.606,Z 603.919,A -85,B 0,C 180,E1 -23046.311,E2 -23046.311} C_VEL
LIN {X 0,Y 320.455,Z 604.608,A -85,B 0,C 180,E1 -23048.801,E2 -23048.801} C_VEL
LIN {X 0,Y 322.929,Z 603.903,A -85,B 0,C 180,E1 -23051.257,E2 -23051.257} C_VEL
LIN {X 0,Y 326.255,Z 601.74,A -85,B 0,C 180,E1 -23053.66,E2 -23053.66} C_VEL
LIN {X 0,Y 329.852,Z 598.172,A -85,B 0,C 180,E1 -23056.025,E2 -23056.025} C_VEL
LIN {X 0,Y 333.858,Z 593.034,A -85,B 0,C 180,E1 -23058.343,E2 -23058.343} C_VEL
LIN {X 0,Y 338.367,Z 586.231,A -85,B 0,C 180,E1 -23060.604,E2 -23060.604} C_VEL
LIN {X 0,Y 342.657,Z 578.777,A -85,B 0,C 180,E1 -23062.526,E2 -23062.526} C_VEL
LIN {X 0,Y 346.619,Z 570.95,A -85,B 0,C 180,E1 -23064.155,E2 -23064.155} C_VEL
LIN {X 0,Y 350.874,Z 561.51,A -85,B 0,C 180,E1 -23065.734,E2 -23065.734} C_VEL
LIN {X 0,Y 355.329,Z 550.346,A -85,B 0,C 180,E1 -23067.278,E2 -23067.278} C_VEL
LIN {X 0,Y 359.206,Z 539.106,A -85,B 0,C 180,E1 -23068.538,E2 -23068.538} C_VEL
LIN {X 0,Y 363.496,Z 524.105,A -85,B 0,C 180,E1 -23069.907,E2 -23069.907} C_VEL
LIN {X 0,Y 366.292,Z 512.309,A -85,B 0,C 180,E1 -23070.765,E2 -23070.765} C_VEL
LIN {X 0,Y 368.832,Z 498.757,A -85,B 0,C 180,E1 -23071.563,E2 -23071.563} C_VEL
LIN {X 0,Y 372.045,Z 477.055,A -85,B 0,C 180,E1 -23072.509,E2 -23072.509} C_VEL
LIN {X 0,Y 378.678,Z 437.011,A -85,B 0,C 180,E1 -23073.906,E2 -23073.906} C_VEL
LIN {X 0,Y 376.42,Z 432.111,A -85,B 0,C 180,E1 -23075.359,E2 -23075.359} C_VEL
LIN {X 0,Y 374.863,Z 428.972,A -85,B 0,C 180,E1 -23076.537,E2 -23076.537} C_VEL
LIN {X 0,Y 373.763,Z 426.634,A -85,B 0,C 180,E1 -23077.524,E2 -23077.524} C_VEL
LIN {X 0,Y 372.084,Z 423.234,A -85,B 0,C 180,E1 -23079.482,E2 -23079.482} C_VEL
LIN {X 0,Y 370.718,Z 421.832,A -85,B 0,C 180,E1 -23081.842,E2 -23081.842} C_VEL
LIN {X 0,Y 370.552,Z 421.626,A -85,B 0,C 180,E1 -23084.379,E2 -23084.379} C_VEL
LIN {X 0,Y 371.872,Z 423.369,A -85,B 0,C 180,E1 -23087.306,E2 -23087.306} C_VEL
LIN {X 0,Y 373.317,Z 426.696,A -85,B 0,C 180,E1 -23089.139,E2 -23089.139} C_VEL
LIN {X 0,Y 373.548,Z 431.934,A -85,B 0,C 180,E1 -23090.097,E2 -23090.097} C_VEL
LIN {X 0,Y 374.007,Z 439.193,A -85,B 0,C 180,E1 -23091.313,E2 -23091.313} C_VEL
LIN {X 0,Y 372.936,Z 456.113,A -85,B 0,C 180,E1 -23092.788,E2 -23092.788} C_VEL
LIN {X 0,Y 371.84,Z 473.903,A -85,B 0,C 180,E1 -23094.148,E2 -23094.148} C_VEL
LIN {X 0,Y 371.037,Z 485.493,A -85,B 0,C 180,E1 -23094.902,E2 -23094.902} C_VEL
LIN {X 0,Y 369.988,Z 495.745,A -85,B 0,C 180,E1 -23095.448,E2 -23095.448} C_VEL
LIN {X 0,Y 363.852,Z 533.706,A -85,B 0,C 180,E1 -23096.808,E2 -23096.808} C_VEL
LIN {X 0,Y 359.982,Z 550.586,A -85,B 0,C 180,E1 -23097.567,E2 -23097.567} C_VEL
LIN {X 0,Y 355.344,Z 566.488,A -85,B 0,C 180,E1 -23098.509,E2 -23098.509} C_VEL
LIN {X 0,Y 350.765,Z 580.309,A -85,B 0,C 180,E1 -23099.554,E2 -23099.554} C_VEL
LIN {X 0,Y 345.472,Z 594.14,A -85,B 0,C 180,E1 -23100.882,E2 -23100.882} C_VEL
LIN {X 0,Y 340.184,Z 606.735,A -85,B 0,C 180,E1 -23102.401,E2 -23102.401} C_VEL
LIN {X 0,Y 335.42,Z 617.35,A -85,B 0,C 180,E1 -23103.989,E2 -23103.989} C_VEL
LIN {X 0,Y 330.546,Z 627.654,A -85,B 0,C 180,E1 -23105.926,E2 -23105.926} C_VEL
LIN {X 0,Y 326.398,Z 636.314,A -85,B 0,C 180,E1 -23107.942,E2 -23107.942} C_VEL
LIN {X 0,Y 322.226,Z 644.435,A -85,B 0,C 180,E1 -23110.31,E2 -23110.31} C_VEL
LIN {X 0,Y 319.097,Z 650.94,A -85,B 0,C 180,E1 -23112.762,E2 -23112.762} C_VEL
LIN {X 0,Y 316.919,Z 655.918,A -85,B 0,C 180,E1 -23115.275,E2 -23115.275} C_VEL
LIN {X 0,Y 315.631,Z 659.201,A -85,B 0,C 180,E1 -23117.538,E2 -23117.538} C_VEL
LIN {X 0,Y 315.202,Z 661.369,A -85,B 0,C 180,E1 -23119.638,E2 -23119.638} C_VEL
LIN {X 0,Y 314.815,Z 670.351,A -85,B 0,C 180,E1 -23121.362,E2 -23121.362} C_VEL
LIN {X 0,Y 314.517,Z 678.723,A -85,B 0,C 180,E1 -23123.285,E2 -23123.285} C_VEL
LIN {X 0,Y 314.367,Z 686.694,A -85,B 0,C 180,E1 -23125.527,E2 -23125.527} C_VEL
LIN {X 0,Y 314.222,Z 692.171,A -85,B 0,C 180,E1 -23127.445,E2 -23127.445} C_VEL
LIN {X 0,Y 314.181,Z 696.601,A -85,B 0,C 180,E1 -23129.361,E2 -23129.361} C_VEL
LIN {X 0,Y 314.031,Z 700.063,A -85,B 0,C 180,E1 -23131.278,E2 -23131.278} C_VEL
LIN {X 0,Y 314.022,Z 703.291,A -85,B 0,C 180,E1 -23133.837,E2 -23133.837} C_VEL
LIN {X 0,Y 314.382,Z 705.095,A -85,B 0,C 180,E1 -23136.396,E2 -23136.396} C_VEL
LIN {X 0,Y 315.2,Z 705.542,A -85,B 0,C 180,E1 -23138.949,E2 -23138.949} C_VEL
LIN {X 0,Y 316.718,Z 704.642,A -85,B 0,C 180,E1 -23141.481,E2 -23141.481} C_VEL
LIN {X 0,Y 319.026,Z 702.39,A -85,B 0,C 180,E1 -23143.976,E2 -23143.976} C_VEL
LIN {X 0,Y 321.877,Z 698.765,A -85,B 0,C 180,E1 -23146.433,E2 -23146.433} C_VEL
LIN {X 0,Y 324.296,Z 695.125,A -85,B 0,C 180,E1 -23148.251,E2 -23148.251} C_VEL
LIN {X 0,Y 328.332,Z 688.839,A -85,B 0,C 180,E1 -23150.61,E2 -23150.61} C_VEL
LIN {X 0,Y 332.446,Z 681.944,A -85,B 0,C 180,E1 -23152.614,E2 -23152.614} C_VEL
LIN {X 0,Y 336.991,Z 673.559,A -85,B 0,C 180,E1 -23154.564,E2 -23154.564} C_VEL
LIN {X 0,Y 342.056,Z 663.414,A -85,B 0,C 180,E1 -23156.448,E2 -23156.448} C_VEL
